(* CODESYS project ATACOMxxxxx_3.0.0.project

Project tree, tasks and I/O mapping:
  Device : HY-TTC 580, TTControl, order no. n/a, version 1.7.1.0
    application Application
      libraries: Standard, * (System); CAA Can Low Level Extern, * (CAA Technical Workgroup); Util, * (System); SysTypes2 Interfaces, * (System); SysTarget, 3.5.5.0 (System); VisuDialogs, * (System); CAA Memory, 3.5.12.0 (CAA Technical Workgroup); Network, 3.5.7.0 (3S - Smart Software Solutions GmbH); lib500, 1.7.1.0 (TTControl); lib500_types, 1.7.1.0 (TTControl); lib500_syscom, 1.7.1.0 (TTControl)
      task _NotificationCallback (externalevent, external event NotificationCallback, priority 0) calls _NotificationCB_PRG
      task _ErrorCallback (externalevent, external event ErrorCallback, priority 1) calls _ErrorCB_PRG
      task CommunicationTask (cyclic, interval t#10ms, priority 31, watchdog t#200ms x 1) calls manageGrCommAndEEPROM, CanCommunication
      task MainTask (cyclic, interval t#10ms, priority 2, watchdog t#200ms x 1) calls MAIN
      Variable lists/
        global variables system
        global variables GVL
        global variables IO
        global variables fieldbus
        global variables par
        global variables CONST
        global variables ERR
        global variables varInput
        global variables display
        global variables ui
        global variables varOutput
      Program logic/
        program _ErrorCB_PRG [ST]
        program _NotificationCB_PRG [ST]
        Tasks/
          program MAIN [ST]: mainLoop, postrun, shutdown, checkParameters, setupCanbus
          program manageGrCommAndEEPROM [ST]: setVariablesToGrComm, initializeGrCommVariables, initializeEepromStructures
          program MachineLogic_PRG [ST]: Cab_C002080
          program CanCommunication [ST]: sendData_to_PC, reciveData_from_PC, initialize
        function initializeCanbus [ST]
        program mngCanbusStatus [ST]: checkCanBusStatus
        program UI_PRG [ST]
        TypeApplication/
          data type Gear9500
      STRUCTURES/
        data type EEPROM_FLAG
        data type CanHandleStatus
        data type MACHINE_MODEL
      Modules/
        IOs/
          Functions/
            program io_module [ST]: instantiateDI, instantiatePWM, instantiatePower, instantiateVOUT, instantiateADC, getInputs, instantiatePWD, initializeIO, instantiateDO, instantiateDIO, instantiatePVG, setOutputs, mngErrors
          program initializeIO [ST]: instantiateAnalogInputs, instantiatePVGOutputs, instantiateDigitalOutputs, instantiateVoltageOutputs, instantiatePWDInputs, instantiatePowerStages, instantiatePWMOutputs, instantiateDigitalInputs
          Types/
            data type pinPWM
            data type type_powerStages
            data type pinADC
            data type type_digitalInputs
            data type pinPVG
            data type type_pwmOutputs
            data type pinPWD
            data type type_voltageOutputs
            data type pinDIO
            data type pwdReadMode
            data type type_digitalOutputs
            data type type_analogInputs
            data type type_pwdInputs
            data type type_pvgOutputs
            data type pin
            data type pinPower
            data type pinVOUT
          global variables sysIO
        COMM/
          Functions/
            program mngCommCan [ST]: mngInit, catchMessages, mngMessage, mngResponse, getsetVarCallback, applyToRamCallback, readAllFromEEPROMCallback, writeToEEPROMCallback, applyToRAM, isVariableValid, initializeVariable
          Types/
            data type grCommVar
            data type grCommAccessRight
            data type grCommVariableStatus
            data type grCommMessageType
            data type grCommEEPROMStatus
          Variable lists/
            global variables grComm
        Canbus/
          Safety interface/
            Tasks/
              program CAN_PRG_SAFE [ST]: exchangeVariables
              program CAN_PRG_UNSAFE [ST]
            Functions/
              program safeSendMessage [ST]
              program safetyCanbusInterface [ST]
              program safeRegisterReceiveMask [ST]
          Variable lists/
            global variables canGVL
            global variables canEVL
          Types/
            data type can
            data type canMessage
            data type canReceiveMask
            data type canBus
          Functions/
            function readMessage [ST]
            program checkReceiveMaskInitialization [ST]
            program registerReceiveMask [ST]
            program sendMessage [ST]
            program initializeCanHandle [ST]
            program checkBusState [ST]
        EEPROM/
          Functions/
            program mngEEPROM [ST]: initEEPROM, mngStep, initializeEepromEntry
          Types/
            Parameters/
              data type HWFW_INFO_TIP
            data type eepromEntry
          Variable lists/
            global variables EEPROM
        Utils/
          program Utils [ST]: decrementUINT, bytesToUInt16, toggle, isNaN, updateValueFiltered, bytesToInt16, decrementUDINT, boolToPWMDutyCycle, linearize, bytesToUReal16, bytesToUDInt32, incrementUINT
        J1939/
          program J1939_PRG [ST]: initReceiveMasks, receiveMessage, parseMessage, sendPGNRequests, mngEngineStatus, redirectToDisplay
          global variables J1939
      visualisation Visualization
    CANs : CANs, TTControl, order no. n/a, version 1.7.1.0
      CAN2 : CAN2, TTControl, order no. n/a, version 1.7.1.0
      CAN3 : CAN3, TTControl, order no. n/a, version 1.7.1.0
      CAN0 : CAN0, TTControl, order no. n/a, version 1.7.1.0
          settings: Baudrate = 250
      CAN1 : CAN1, TTControl, order no. n/a, version 1.7.1.0
      CAN6 : CAN6, TTControl, order no. n/a, version 1.7.1.0
      CAN4 : CAN4, TTControl, order no. n/a, version 1.7.1.0
      CAN5 : CAN5, TTControl, order no. n/a, version 1.7.1.0
    System : System, TTControl, order no. n/a, version 1.7.1.0
        unmapped channels: mode, error, mode, error, mode, error, mode, error, mode, error, mode, error, mode, error, shutdown, error, enable_error_group_0, enable_error_group_1, enable_error_group_2, diag_status, safe_state, error, driver_init_error, UBAT, Terminal_15, WakeUp, Temperature, SSW0, SSW1, SSW2, SSUP0, SSUP1, SSUP2, status, write, boot_error, trigger_error, Powerstage, SSW0, SSW1,
          SSW2, SSUP0, SSUP1, SSUP2, Terminal_15, WakeUp, ExtShutOff0, ExtShutOff1, ExtShutOff2
      Timer_Inputs : TIN, TTControl, order no. n/a, version 1.7.1.0
        Pin 147
          <Empty>
        Pin 122
          <Empty>
        Pin 148
          <Empty>
        Pin 146
          <Empty>
        Pin 124
          <Empty>
        Pin 123
          <Empty>
      Analog_Inputs_2Mode_10V : AIN_2Mode_10V, TTControl, order no. n/a, version 1.7.1.0
        Pin 134
          <Vuoto>
        Pin 109
          <Empty>
        Pin 132
          <Vuoto>
        Pin 131
          <Empty>
        Pin 107
          <Vuoto>
        Pin 110
          <Vuoto>
        Pin 108
          <Empty>
        Pin 133
          <Empty>
      Analog_Inputs_3Mode : AIN_3Mode, TTControl, order no. n/a, version 1.7.1.0
        Pin 129
          <Vuoto>
        Pin 104
          <Vuoto>
        Pin 130
          <Vuoto>
        Pin 105
          <Vuoto>
        Pin 103
          <Vuoto>
        Pin 127
          <Vuoto>
        Pin 106
          <Vuoto>
        Pin 128
          <Empty>
      Digital_Outputs_LS : LSDOUT, TTControl, order no. n/a, version 1.7.1.0
        Pin 239
          <Vuoto>
        Pin 251
          <Vuoto>
        Pin 240
          <Vuoto>
        Pin 252
          <Vuoto>
        Pin 254
          <Vuoto>
        Pin 238
          <Vuoto>
        Pin 253
          <Vuoto>
        Pin 241
          <Vuoto>
      Timer_Inputs_Cur : TIN_Cur, TTControl, order no. n/a, version 1.7.1.0
        Pin 140
          <Empty>
        Pin 117
          <Vuoto>
        Pin 116
          <Empty>
        Pin 139
          <Empty>
        Pin 115
          <Vuoto>
        Pin 141
          <Vuoto>
      Analog_Inputs_2Mode_32V : AIN_2Mode_32V, TTControl, order no. n/a, version 1.7.1.0
        Pin 113
          <Empty>
        Pin 137
          <Empty>
        Pin 136
          <Empty>
        Pin 112
          <Empty>
        Pin 138
          <Empty>
        Pin 114
          <Empty>
        Pin 111
          <Vuoto>
        Pin 135
          <Empty>
      PWM_Outputs : PWM, TTControl, order no. n/a, version 1.7.1.0
        Safety_switch_0 : PWM_SSW0, TTControl, order no. n/a, version 1.7.1.0
          Pin 165
            <Empty>
          Pin 195
            <Vuoto>
          Pin 162
            <Empty>
          Pin 171
            <Vuoto>
          Pin 168
            <Empty>
          Pin 186
            <Empty>
          Pin 183
            <Empty>
          Pin 177
            <Vuoto>
          Pin 180
            <Empty>
          Pin 159
            <Empty>
          Pin 153
            <Vuoto>
          Pin 189
            <Empty>
          Pin 156
            <Empty>
          Pin 192
            <Empty>
        Safety_switch_1 : PWM_SSW1, TTControl, order no. n/a, version 1.7.1.0
          Pin 157
            <Empty>
          Pin 187
            <Empty>
          Pin 154
            <Vuoto>
          Pin 160
            <Empty>
          Pin 178
            <Empty>
          Pin 169
            <Vuoto>
          Pin 166
            <Vuoto>
          Pin 163
            <Empty>
          Pin 184
            <Empty>
          Pin 181
            <Empty>
          Pin 190
            <Vuoto>
          Pin 172
            <Vuoto>
          Pin 193
            <Vuoto>
          Pin 196
            <Vuoto>
        Safety_switch_2 : PWM_SSW2, TTControl, order no. n/a, version 1.7.1.0
          Pin 101
            <Vuoto>
          Pin 125
            <Vuoto>
          Pin 150
            <Vuoto>
          Pin 174
            <Vuoto>
          Pin 102
            <Vuoto>
          Pin 126
            <Vuoto>
          Pin 151
            <Vuoto>
          Pin 175
            <Vuoto>
      Digital_Outputs_HS : HSDOUT, TTControl, order no. n/a, version 1.7.1.0
        Pin 176
          <Vuoto>
        Pin 149
          <Vuoto>
        Pin 158
          <Vuoto>
        Pin 173
          <Vuoto>
        Pin 152
          <Vuoto>
        Pin 155
          <Vuoto>
        Pin 182
          <Vuoto>
        Pin 179
          <Vuoto>
      PVG_Outputs : PVG, TTControl, order no. n/a, version 1.7.1.0
        Pin 161
          <Vuoto>
        Pin 185
          <Vuoto>
        Pin 188
          <Vuoto>
        Pin 164
          <Vuoto>
        Pin 191
          <Vuoto>
        Pin 167
          <Vuoto>
        Pin 194
          <Vuoto>
        Pin 170
          <Vuoto>
  text list GlobalTextList
*)

// Device/Application/STRUCTURES/EEPROM_FLAG
TYPE EEPROM_FLAG : //verificata
STRUCT
	READ: BOOL:= FALSE;
	CHANGED: BOOL:= FALSE;
	WRITE: BOOL:= FALSE;
END_STRUCT
END_TYPE

// Device/Application/Modules/COMM/Types/grCommVar
TYPE grCommVar :
	STRUCT;
		accessRights: grCommAccessRight;
		status: grCommVariableStatus;
		
		pointerToSystemVar: POINTER TO UINT;
		uiLowerValidValue: UINT;
		uiHigherValidValue: UINT;
		uiDefaultValue: UINT;
		
		uiValue: UINT;
	END_STRUCT
END_TYPE

// Device/Application/Modules/COMM/Types/grCommAccessRight
{attribute 'qualified_only'}
{attribute 'strict'}
TYPE grCommAccessRight :
(
	NoAccess := 0,
	ReadOnly := 1,
	ReadWrite := 2
);
END_TYPE

// Device/Application/Modules/COMM/Types/grCommVariableStatus
{attribute 'qualified_only'}
{attribute 'strict'}
TYPE grCommVariableStatus :
(
	Uninitialized:= 0,
	Pristine:= 1,
	ModifiedByRemote:= 2,
	Error:= 3
);
END_TYPE

// Device/Application/Modules/COMM/Types/grCommMessageType
{attribute 'qualified_only'}
{attribute 'strict'}
TYPE grCommMessageType :
(
	ExitCode:= 0,				// Esito di un comando
	
	GetVariable:= 1,			// Get valore di una variabile
	SetVariable:= 2,			// Set valore di una variabile
	HeartRateRequest:= 3,		// Richiesta di heart rate (broadcast)
	LoadFromEEPROM:= 4,			// Leggi parametri da EEPROM
	WriteToEEPROM:= 5,			// Scrivi parametri in RAM sulla EEPROM (rispettando il flag EDIT)
	WriteAllToEEPROM:= 6,		// Scrivi parametri in RAM sulla EEPROM (ignorando il flag EDIT)
	ApplyVariables:= 7,			// Imposta i parametri inviati sulla RAM
	
	ErrorCode:= 255		// Errore
);
END_TYPE

// Device/Application/Modules/IOs/Types/pinPWM
TYPE pinPWM EXTENDS pin :
	STRUCT
		stErrorGetCut: lib500_types.IO_ERRORTYPE;
		wFrequency: WORD:= 100;
		bPolarity: BOOL:= TRUE;
		bDiagMargin: BOOL:= FALSE;
		wFeedbackHighTime: WORD;
		wPeriodFeedback: WORD;
		wCurrent: WORD;
		bCurrentFresh: BOOL;
		wDuty: WORD;
	END_STRUCT
END_TYPE

// Device/Application/Modules/IOs/Types/type_powerStages
TYPE type_powerStages :
STRUCT	
	safetySwitch0: pinPower;	
	safetySwitch1: pinPower;	
	safetySwitch2: pinPower;
	powerStage: pinPower;
	sensorSupply0: pinPower;
	sensorSupply1: pinPower;
	sensorSupply2: pinPower;
END_STRUCT
END_TYPE

// Device/Application/Modules/IOs/Types/pinADC
TYPE pinADC EXTENDS pin :
	STRUCT		
		stADCType: lib500_types.IO_ADC_TYPE;
		stADCRange: lib500_types.IO_ADC_RANGE;
		stADCSensorSupply: lib500_types.IO_SENSOR_SUPPLY;
		dwValue: DWORD;
		bValueFresh: BOOL;
	END_STRUCT
END_TYPE

// Device/Application/Modules/COMM/Types/grCommEEPROMStatus
{attribute 'qualified_only'}
{attribute 'strict'}
TYPE grCommEEPROMStatus :
(
	Idle:= 0,
	BeginRead:= 1,
	Reading:= 2,
	BeginWrite:= 3,
	Writing
);
END_TYPE

// Device/Application/Modules/IOs/Types/type_digitalInputs
TYPE type_digitalInputs :
STRUCT	
	fuelReserve_p127: pinDIO;
	alternatorD_p111: pinDIO;
	gearSelectorFwInching_p135: pinDIO;
	gearSelectorFirstSlow_p112: pinDIO;
	gearSelectorBwInching_p136: pinDIO;
	gearSelectorSecondFast_p113: pinDIO;
	inchingSwitch_p137: pinDIO;
	compressedAirSwitch_p114: pinDIO;
	safetySwitch_p138: pinDIO;
	
	parkingBrakeLamp_p140: pinDIO;
	airPressureLowLamp_p177: pinDIO;
	transOilOvertempLamp_p156: pinDIO;
	brakeFluidLowLamp_p180: pinDIO;
	coolantLevelLow_p159: pinDIO;
	
	engineStartK50_p117: pinDIO;
	seatSwitch_p146: pinDIO;
	forwardSwitch_p123: pinDIO;
	backwardSwitch_p147: pinDIO;
	neutralSwitch_p124: pinDIO;
	
	turtleSwitch_p161: pinDIO;
	positionLightsSwitch_p185: pinDIO;
	lowBeamLightsSwitch_p188: pinDIO;
	highBeamFlashLightsSwitch_p164: pinDIO;
	highBeamLightsSwitch_p116: pinDIO;
	leftBlinkerSwitch_p191: pinDIO;
	rightBlinkerSwitch_p167: pinDIO;
	hazardSwitch_p194: pinDIO;
	parkingBrakeSwitchOptional_p170: pinDIO;
	
	speedLimiterSwitch_p129: pinDIO;
	
	gearShiftUp_p122: pinDIO;
	gearShiftDown_p148: pinDIO;
	autoDetect9500_p238: pinDIO;
	
	

	
	input_115: pinDIO;
	input_116: pinDIO;
	input_117: pinDIO;
	input_122: pinDIO;
	input_123: pinDIO;
	input_124: pinDIO;
	input_139: pinDIO;
	input_140: pinDIO;
	input_141: pinDIO;
	input_146: pinDIO;
	input_147: pinDIO;
	input_148: pinDIO;
	input_161: pinDIO;
	input_164: pinDIO;
	input_167: pinDIO;
	input_170: pinDIO;
	input_185: pinDIO;
	input_188: pinDIO;
	input_191: pinDIO;
	input_194: pinDIO;
	
	
	
	
END_STRUCT
END_TYPE

// Device/Application/Modules/IOs/Types/pinPVG
TYPE pinPVG EXTENDS pin :
	STRUCT
		stGetVoltageError: lib500_types.IO_ERRORTYPE;
		wValue: WORD := 5000;
		uiReadVoltage: UINT := 0;
		bVoltageFresh: BOOL := FALSE;
	END_STRUCT
END_TYPE

// Device/Application/Modules/Canbus/Types/can
TYPE can :
	STRUCT
			
		bInitialized: BOOL:= FALSE;	
		usiChannel: USINT:= 0;
		uiBaudrateKbps: UINT:= 0;
	
		driver: CL2.CAA.HANDLE;
		initializeError: CL2.ERROR;
		transmitError: CL2.ERROR;
		busStatus: CL2.BUSSTATE;
		
		receiveMessageHandle: CL2.CAA.HANDLE := CL2.CAA.gc_hINVALID;
		pointerToData: POINTER TO CL2.CL2I.DATA;
		messageLeft : CL2.CAA.COUNT;
		
		uiMessageCount: INT:=0;
		byaReceiveBuffer: ARRAY [0..7] OF BYTE;				
		byaTransmitBuffer: ARRAY [0..7] OF BYTE;						
		
	END_STRUCT
END_TYPE

// Device/Application/Modules/IOs/Types/type_pwmOutputs
TYPE type_pwmOutputs :
STRUCT
	turtleBtnBacklight_p168: pinPWM;
	hazardBtnBacklight_p190: pinPWM;
END_STRUCT
END_TYPE

// Device/Application/Modules/Canbus/Types/canMessage
TYPE canMessage :
	STRUCT
		udiId: UDINT:= 0;
		bExtended: BOOL:= FALSE;
		byLength: BYTE:= 8;
		byaData: ARRAY [0..7] OF BYTE;
	END_STRUCT
END_TYPE

// Device/Application/Modules/Canbus/Types/canReceiveMask
TYPE canReceiveMask :
	STRUCT
		bActive: BOOL:= FALSE;
		bInitialized: BOOL:= FALSE;
		udiId: UDINT:= 0;
		stCAAMask: CL2.CAA.HANDLE:= CL2.CAA.gc_hINVALID;	
		stMessagesLeft: CL2.CAA.COUNT;	
		udiCobIdMask: UDINT:= 16#1FFFFFFF;
	END_STRUCT
END_TYPE

// Device/Application/Modules/Canbus/Types/canBus
TYPE canBus :
	STRUCT
		bActive: BOOL:= FALSE;
		stChannel: can;
		staReceiveMasks: ARRAY[0..canGVL.iReceiveMaskCount-1] OF canReceiveMask;
		stTransmitBuffer: ARRAY[0..canGVL.iTransmitBufferSize-1] OF canMessage;
	END_STRUCT
END_TYPE

// Device/Application/Modules/IOs/Types/pinPWD
TYPE pinPWD EXTENDS pin :
	STRUCT
		stGetVoltageError: lib500_types.IO_ERRORTYPE;
		stIncSetError: lib500_types.IO_ERRORTYPE;
		pwdMode: lib500_types.IO_PWD_INC_MODE;
		wCountInit: WORD:= 32767;
		wCount: WORD;
		wCountZero: WORD;
		uiVoltage: UINT;
		bChannelA: BOOL;
		bChannelB: BOOL;
		readMode: pwdReadMode;
		pulseSamples: lib500_types.IO_PWD_PULSE_SAMPLES;
		dwFrequencyHz: DWORD;
		dwPulseWidth: DWORD;
		pulseMode: lib500_types.IO_PWD_PULSE_MODE;
		freqMode: lib500_types.IO_PWD_FREQ_MODE;
		byCaptureCount: BYTE;
		bVoltageFresh: BOOL;
		bSetIncrementCount: BOOL:= FALSE;
	END_STRUCT
END_TYPE

// Device/Application/Modules/IOs/Types/type_voltageOutputs
TYPE type_voltageOutputs :
STRUCT
	// dummy: pinVOUT;
END_STRUCT
END_TYPE

// Device/Application/STRUCTURES/CanHandleStatus
TYPE CanHandleStatus :
	STRUCT
		uidFreeMessagesInPoll: UDINT:= 0;
		uidMessagesInElabQueue: UDINT:= 0;
	END_STRUCT
END_TYPE

// Device/Application/Modules/IOs/Types/pinDIO
TYPE pinDIO EXTENDS pin :
	STRUCT
		bValue: BOOL:= FALSE;
		wCurrent: WORD;
		bCurrentFresh: BOOL;
		stErrorGetCut: lib500_types.IO_ERRORTYPE;
	END_STRUCT
END_TYPE

// Device/Application/Modules/IOs/Types/pwdReadMode
{attribute 'qualified_only'}
{attribute 'strict'}
TYPE pwdReadMode :
(
	incremental := 0,
	complex
);
END_TYPE

// Device/Application/Modules/IOs/Types/type_digitalOutputs
TYPE type_digitalOutputs :
STRUCT				 
	lampeggiante_p183: pinDIO;
	workLights_p186: pinDIO;
	airCompressorRelay_p162: pinDIO;
	dashboardBacklight_p189: pinDIO;
	workModeActiveDpfLamp_p165: pinDIO;
	forwardGearEV_p192: pinDIO;

	backwardGearEV_p193: pinDIO;
		
	highBeamLights_p149: pinDIO;
	highBeamLights_p173: pinDIO;
	
	lowBeamLights_p152: pinDIO;
	lowBeamLights_p176: pinDIO;
	
	positionLights_p155: pinDIO;
	positionLights_p179: pinDIO;
	
	inchingBrakeEV_p171: pinDIO;
	parkingBrakeEV_p154: pinDIO;
	pneumaticParkBrakeEV_p178: pinDIO;
	rightBlinker_p157: pinDIO;
	leftBlinker_p181: pinDIO;
	reverseLight_p160: pinDIO;
	neutralGear_p254: pinDIO;
	reverseBuzzer_p184: pinDIO;
	
	inchingLamp_p163: pinDIO;
	daytimeLights_p187: pinDIO;
	displayK15_p166: pinDIO;
	
	slowGearEV_p195: pinDIO;//gearEvC_p195: pinDIO;
	gearEvD_p169: pinDIO;
	gearEvE_p196: pinDIO;
	
	output_149: pinDIO;
	output_150: pinDIO;
	output_152: pinDIO;
	output_153: pinDIO;
	output_154: pinDIO;
	output_155: pinDIO;
	output_156: pinDIO;
	output_157: pinDIO;
	output_158: pinDIO;
	output_159: pinDIO;
	output_173: pinDIO;
	output_174: pinDIO;
	output_176: pinDIO;
	output_177: pinDIO;
	output_178: pinDIO;
	output_179: pinDIO;
	output_180: pinDIO;
	output_181: pinDIO;
	output_182: pinDIO;
	output_183: pinDIO;
END_STRUCT
END_TYPE

// Device/Application/Modules/IOs/Types/type_analogInputs
TYPE type_analogInputs :
STRUCT
	ecuK15_p207: pinADC;
	fuelTankGauge_p103: pinADC;	
	pneumaticTankGauge_p104: pinADC;
	shiftOilGauge_p128: pinADC;	
	
	speedLimiterReduction_p251: pinADC;	
END_STRUCT
END_TYPE

// Device/Application/Modules/IOs/Types/type_pwdInputs
TYPE type_pwdInputs :
STRUCT
	//speedSensor_p115: pinPWD;
	transmissionShaftSensor5000_p175: pinPWD;
	transmissionShaftSensor7500_p151: pinPWD;
END_STRUCT
END_TYPE

// Device/Application/Modules/IOs/Types/type_pvgOutputs
TYPE type_pvgOutputs :
STRUCT
	//_p161: pinPWD;
END_STRUCT
END_TYPE

// Device/Application/Modules/IOs/Types/pin
TYPE pin :
	STRUCT
		bInitialized: BOOL:= FALSE;
		stInitError: lib500_types.IO_ERRORTYPE;
		stError: lib500_types.IO_ERRORTYPE;
		byChannel: BYTE;
		byPullType: BYTE;
		byMinTTCModel: BYTE:= 0;
		byResetCount: BYTE:= 0;
	END_STRUCT
END_TYPE

// Device/Application/Modules/IOs/Types/pinPower
TYPE pinPower EXTENDS pin :
	STRUCT
		mode: lib500_types.IO_POWER_STATE;
	END_STRUCT
END_TYPE

// Device/Application/Modules/EEPROM/Types/eepromEntry
TYPE eepromEntry :
	STRUCT
		wAddress: WORD;
		pData: POINTER TO BYTE;
		wSize: WORD;
	END_STRUCT
END_TYPE

// Device/Application/Modules/EEPROM/Types/Parameters/HWFW_INFO_TIP
TYPE HWFW_INFO_TIP :
	STRUCT		
		PASSWORD_LEVEL_0: UINT:= 0;
		PASSWORD_LEVEL_1: UINT:= 1234;		
	END_STRUCT
END_TYPE

// Device/Application/Modules/IOs/Types/pinVOUT
TYPE pinVOUT EXTENDS pin :
	STRUCT
		wOutputVoltageMv: WORD:= 0;
	END_STRUCT
END_TYPE

// Device/Application/STRUCTURES/MACHINE_MODEL
{attribute 'qualified_only'}
{attribute 'strict'}
TYPE MACHINE_MODEL :
(
	ATA_5000 := 0,
	ATA_7500,
	ATA_9500
);
END_TYPE

// Device/Application/Program logic/TypeApplication/Gear9500
{attribute 'qualified_only'}
{attribute 'strict'}
TYPE Gear9500 :
(
	GEAR_1ST := 1,
	GEAR_2ND,
	GEAR_3RD,
	GEAR_4TH
);
END_TYPE

// Device/Application/Modules/COMM/Variable lists/grComm
{attribute 'qualified_only'}

(* User code configurable settings *)
VAR_GLOBAL CONSTANT
	uiProtocolMessageID : UINT:=16#7F7;
	uiProtocolVirtualNode : UINT:=16#3;	
	uiVariablesMaxIndex: UINT:= 100;    // Reduce this value if you have low memory issues
END_VAR



(* User code accessible status variables *)
VAR_GLOBAL  			
	bCommunicationActive: BOOL:=FALSE;			// Indicates that a communication is running
	bTriggerReadFromEEPROM: BOOL:= TRUE;		// If active user code should read variables from EEPROM and store their value in grComm.staVariables
	bTriggerApplyToRAM: BOOL:= FALSE;			// If active user code should set its system values from grComm.staVariables
	bTriggerWriteToEEPROM: BOOL:= FALSE;		// If active user code should write to EEPROM only the modified variable's values from grComm.staVariables
	bTriggerWriteAllToEEPROM: BOOL:= FALSE;		// If active user code should write to EEPROM all the variable's values from grComm.staVariables
END_VAR


(* Internal logic variables *)
VAR_GLOBAL
	staVariables: ARRAY[1..uiVariablesMaxIndex] OF grCommVar;	
END_VAR

(* Internal logic defines *)
VAR_GLOBAL CONSTANT	
	COMM_TIMER_RLD: UINT:= 1000;
	LIB_VERSION_CODE: BYTE:= 0;		
	
	// Exit code viene messo nel campo ADDRESS se TYPE == EXIT_CODE
	EXIT_CODE_ERROR: UINT:= 0;
	EXIT_CODE_OK: UINT:= 1;

END_VAR

// Device/Application/Variable lists/system
{attribute 'qualified_only'}
VAR_GLOBAL CONSTANT	
	FWV_PRIMARIA: BYTE:=0;
	FWV_SECONDARIA: BYTE:=0;
	FWV_BUGFIX: BYTE:=0;	
END_VAR

VAR_GLOBAL	
	xFirstCycle: BOOL:= TRUE;
	
	machineModel: MACHINE_MODEL;
	
	fwVMergedPrimarySecondary: UINT:= (FWV_PRIMARIA * 256) OR FWV_SECONDARIA;
	fwVMergedRevisionBugfix: UINT:= FWV_BUGFIX;
	bHasAlarms: BOOL:= FALSE;	
	
	matricolaL: UINT:= 0;
	matricolaH: UINT:= 0;
	
	bParametersReady: BOOL:= FALSE;	
	systemAlarms: UINT:= 0;
	
	xHazardStatus: BOOL:= FALSE;
	xParkingBrakeActive: BOOL:= FALSE;
	xParkingBrakeLampInputActive: BOOL:= FALSE;
	xInchingModeActive: BOOL:= FALSE;
	
	byActiveGear: BYTE:= 0;  (* 1-EvMarciaLentaAttiva, 2-EvMarciaLentaDisattiva NoInching, 3-Inching  *)
	byDirection: BYTE:= 0;  (* 0- ferma, 1-avanti, 2 indietro *)
	byFuelPercent: BYTE;
	
	xSeatStatus: BOOL;
	rFuelLevelFiltered: REAL;
	udiInchingAlertTimerMs: UDINT;
	
	rSpeedKmph: REAL;
	xIncorrectStart: BOOL;
END_VAR

// Device/Application/Variable lists/GVL
{attribute 'qualified_only'}
VAR_GLOBAL
	MODELLO_CENTRALINA: BYTE;
	fwVersion: ARRAY[0..2] OF BYTE:= [3, 0, 0];  // versione di cenrtralina 3.0.0
	
	xAllowSystemShutdown: BOOL;
	xDPFRegenerationRequestInput: BOOL;	
	xSpeedLimitStatus: BOOL:= FALSE;
END_VAR

// Device/Application/Variable lists/IO
{attribute 'qualified_only'}
VAR_GLOBAL
	xECUK15: BOOL;
	
	xSpeedLimFromAdc: BOOL;
END_VAR

// Device/Application/Modules/Canbus/Variable lists/canGVL
{attribute 'qualified_only'}

VAR_GLOBAL CONSTANT	
	iBusCount: INT:= 10;
	iTransmitBufferSize: INT:= 50;
	iReceiveMaskCount: INT:= 50;
END_VAR

VAR_GLOBAL
	busses: ARRAY[0..iBusCount-1] OF canBus;
END_VAR

// Device/Application/Variable lists/fieldbus
{attribute 'qualified_only'}
VAR_GLOBAL CONSTANT
	iCanbusCount: INT:= 4;
	uiaCanBaudrates: ARRAY[0..9] OF UINT:= [500, 250, 250, 0, 0, 0, 0, 0, 0, 0];
END_VAR

VAR_GLOBAL
	can: ARRAY [0..9] OF canBus;
	
	bCanbusInitialized: BOOL:= FALSE;
END_VAR

// Device/Application/Variable lists/par
{attribute 'qualified_only'}
VAR_GLOBAL
	stHwFwInfo: HWFW_INFO_TIP;
END_VAR

// Device/Application/Variable lists/CONST
{attribute 'qualified_only'}
VAR_GLOBAL	
	CANBUS_MAX_READS_PER_CYCLE: BYTE:= 10;
	CANBUS_MIN_FREE_POLL: BYTE:= 30;
	CANBUS_MAX_RX_QUEUE: BYTE:= 15;
END_VAR

// Device/Application/Modules/IOs/sysIO
{attribute 'qualified_only'}
VAR_GLOBAL
	bIOInstantiated: BOOL:= FALSE;
	bIOInitialized: BOOL:= FALSE;

	digitalInput: type_digitalInputs;
	analogInput: type_analogInputs;
	pwdInput: type_pwdInputs;
	pvgOutput: type_pvgOutputs;
	
	digitalOutput: type_digitalOutputs;
	powerStage: type_powerStages;
	pwmOutput: type_pwmOutputs;
	voltageOutput: type_voltageOutputs;
END_VAR

// Device/Application/Modules/Canbus/Variable lists/canEVL
(* THIS EVL IS AUTOGENERATED. DO NOT MODIFY THESE ATTRIBUTES. *)
{attribute 'location' := '16#800' }
{attribute 'linkalways'}
{attribute 'qualified_only'}
VAR_GLOBAL	
	bHasChanges: BOOL:= FALSE;
	bChannelsHasChanges: BOOL:= FALSE;
	bTransmitBuffersHasChanges: BOOL:= FALSE;
	bMasksHasChanges: BOOL:= FALSE;
	busses: ARRAY[0..canGVL.iBusCount-1] OF canBus;
END_VAR

// Device/Application/Modules/EEPROM/Variable lists/EEPROM
{attribute 'qualified_only'}

(* User code accessible status indicators *)
VAR_GLOBAL
	bTriggerReadAll: BOOL:= FALSE;
	
	bEEPROMInitialized: BOOL := FALSE;
	bReadFromEEPROM: BOOL := TRUE;
	bWriteAllToEEPROM: BOOL:= FALSE;
END_VAR


(* Internal logic *)
VAR_GLOBAL CONSTANT	
	iEepromEntriesCount: INT:= 160;
END_VAR
VAR_GLOBAL	
	staAllEntries: ARRAY[0..iEepromEntriesCount-1] OF eepromEntry; // On TTC-500 series EEPROM is 64KB. Each structure has 400 byte of space reserved
END_VAR

// Device/Application/Variable lists/ERR
{attribute 'qualified_only'}
VAR_GLOBAL
	xInputPins: BOOL;
	xOutputPins: BOOL;
	xInitializePins: BOOL;
	xCanbusHeavy: BOOL;
END_VAR

// Device/Application/Variable lists/varInput
{attribute 'qualified_only'}
VAR_GLOBAL
	xInput_1: BOOL;
	xInput_2: BOOL;
	xInput_3: BOOL;
	xInput_4: BOOL;
	xInput_5: BOOL;
	xInput_6: BOOL;
	xInput_7: BOOL;
	xInput_8: BOOL;
	xInput_9: BOOL;
	xInput_10: BOOL;
	xInput_11: BOOL;
	xInput_12: BOOL;
	xInput_13: BOOL;
	xInput_14: BOOL;
	xInput_15: BOOL;
	xInput_16: BOOL;
	xInput_17: BOOL;
	xInput_18: BOOL;
	xInput_19: BOOL;
	xInput_20: BOOL;
END_VAR

// Device/Application/Variable lists/display
{attribute 'qualified_only'}
VAR_GLOBAL
	xLampeggianteOffStatus: BOOL:= FALSE;
	xWorkLightStatus: BOOL:= FALSE;
	xDRLOffStatus: BOOL:= FALSE;
	xSpeedLimitRequest: BOOL:= FALSE;
	
	xInput1, xInput2, xInput3, xInput4, xInput5, xInput6, xInput7, xInput8: BOOL;
END_VAR

// Device/Application/Variable lists/ui
{attribute 'qualified_only'}
VAR_GLOBAL
	xBlinker_100ms: BOOL;
	xBlinker_500ms: BOOL;
END_VAR

// Device/Application/Modules/J1939/J1939
{attribute 'qualified_only'}
VAR_GLOBAL
	byECUNodeId: BYTE:= 16#10;
	xEngineOnline: BOOL:= FALSE;
	xSendPGNRequest: BOOL:= FALSE;
	xRedirectMessages: BOOL:= FALSE;
	
	// valori in arrivo dal bus
	iTorquePercent: INT;
	uiEngineSpeedRpm: UINT;
	uiMinutesRunWhileMILAct: UINT;
	lrEngineTotalFuelUsedLiters: LREAL;
	rEngineFuelRateLph: REAL;
	byBarometricPressureKPa: BYTE;
	iAmbientAirTemperatureDegC: INT;
	iEngineIntakeAirTemperatureDegC: INT;
	uiOilPressureKPa: UINT;
	byCoolantLevelPerc: BYTE;
	iEngineCoolantTempDegC: INT;
	iEngineFuelTempDegC: INT;
	iAftertreatmentDPFIntakeGasTempDegC: INT;
	rBatteryPotentialV: REAL;
	byEngineStartEnable: BYTE;
	rEngineTotalIdleHours: REAL;
	byAftertreatmentEngineSpeedIncreaseRequest: BYTE;
	byEngineWaitToStartLamp: BYTE;
	byEngineIdleShutdownStatus: BYTE;
	byEngineIdleShutdownAlert: BYTE;
	byServiceComponentId1: BYTE;
	byServiceComponentId2: BYTE;
	byServiceComponentId3: BYTE;
	iServiceDelayHours: INT;
	rEngineTotalOperationHours: REAL;
	byDPFFilterLamp: BYTE;
	byAftertreatmentDPFActiveRegeneration: BYTE;
	byAftertreatmentDPFFilterStatus: BYTE;
	byDPFActiveRegenerationInhibitedDueSwitch: BYTE;
	byDPFActiveRegenerationInhibitedDueTmpSysLock: BYTE;
	byDPFActiveRegenerationInhibitedDuePermSysLock: BYTE;
	
	
	byWarningIndicator: BYTE;	
	byWarningIndicatorFlash: BYTE;
	byShutdownIndicator: BYTE;
	byEngineProtectIndicator: BYTE;
	byEngineProtectIndicatorFlash: BYTE;
	byEmissionSystemMalfunctionIndicator: BYTE;
	byEmissionSystemMalfunctionIndicatorFlash: BYTE;	
	
	
	// trouble codes
	DM1_SPN: ULINT;
	DM1_FMI: UINT;
	DM1_OC: UINT;
	
	
	// valori calcolati
	xEngineRunning: BOOL;
	xEngineDPFRegenRequest: BOOL;
	xEngineDPFRegenActive: BOOL;
	xLowOilPressure: BOOL;
	xEngineLamp: BOOL;
	xEngineLampRed: BOOL;
	byRegenerationStatus: BYTE;
	
	
END_VAR

// Device/Application/Variable lists/varOutput
{attribute 'qualified_only'}
VAR_GLOBAL
	xOutput_1: BOOL;
	xOutput_2: BOOL;
	xOutput_3: BOOL;
	xOutput_4: BOOL;
	xOutput_5: BOOL;
	xOutput_6: BOOL;
	xOutput_7: BOOL;
	xOutput_8: BOOL;
	xOutput_9: BOOL;
	xOutput_10: BOOL;
	xOutput_11: BOOL;
	xOutput_12: BOOL;
	xOutput_13: BOOL;
	xOutput_14: BOOL;
	xOutput_15: BOOL;
	xOutput_16: BOOL;
	xOutput_17: BOOL;
	xOutput_18: BOOL;
	xOutput_19: BOOL;
	xOutput_20: BOOL;
END_VAR

// Device/Application/Program logic/_NotificationCB_PRG
PROGRAM _NotificationCB_PRG
VAR
	diag_state : lib500_types.DIAG_STATETYPE := lib500_types.DIAG_STATETYPE.DIAG_STATE_DISABLED;
	watchdog_state : lib500_types.DIAG_WD_STATETYPE := lib500_types.DIAG_WD_STATETYPE.DIAG_WD_STATE_UNKNOWN;
	error : lib500_types.DIAG_ERRORCODE := (error_code := lib500_types.DIAG_ERRORTYPE.DIAG_E_NOERROR, 
                                            device_num := lib500_types.DIAG_DEVICETYPE.DIAG_DEV_NONE,
                                            faulty_value := 0);
	return_code : lib500_types.IO_ERRORTYPE := lib500_types.IO_ERRORTYPE.IO_E_UNKNOWN;
	
	call_count : UDINT := 0;
END_VAR

(* get the reason for the notification callback *)
return_code := lib500.DIAG_CDS_GetNotificationReason(ADR(diag_state), 
                                                     ADR(watchdog_state),
                                                     ADR(error));

(* custom handler code can be placed here *)

(* increment call count *)
call_count := call_count + 1;

END_PROGRAM

// Device/Application/Program logic/_ErrorCB_PRG
PROGRAM _ErrorCB_PRG
VAR
	diag_state : lib500_types.DIAG_STATETYPE := lib500_types.DIAG_STATETYPE.DIAG_STATE_DISABLED;
	watchdog_state : lib500_types.DIAG_WD_STATETYPE := lib500_types.DIAG_WD_STATETYPE.DIAG_WD_STATE_UNKNOWN;
	error : lib500_types.DIAG_ERRORCODE := (error_code := lib500_types.DIAG_ERRORTYPE.DIAG_E_NOERROR, 
                                            device_num := lib500_types.DIAG_DEVICETYPE.DIAG_DEV_NONE,
                                            faulty_value := 0);
	return_code : lib500_types.IO_ERRORTYPE := lib500_types.IO_ERRORTYPE.IO_E_UNKNOWN;
	
	reaction : lib500_types.DIAG_REACTION := lib500_types.DIAG_REACTION.DIAG_ERR_SAFESTATE;
	
	call_count : UDINT := 0;
END_VAR

(* get the reason for the error callback *)
return_code := lib500.DIAG_CDS_GetErrorReason(ADR(diag_state), 
                                              ADR(watchdog_state),
                                              ADR(error));

(* custom handler code can be placed here *)

(* the choices for the reactions are:
   -> lib500_types.DIAG_REACTION.DIAG_ERR_NOACTION
   -> lib500_types.DIAG_REACTION.DIAG_ERR_SAFESTATE
   -> lib500_types.DIAG_REACTION.DIAG_ERR_DISABLE_SSW0
   -> lib500_types.DIAG_REACTION.DIAG_ERR_DISABLE_SSW1
   -> lib500_types.DIAG_REACTION.DIAG_ERR_DISABLE_SSW2
   -> lib500_types.DIAG_REACTION.DIAG_ERR_DISABLE_HS00
   -> lib500_types.DIAG_REACTION.DIAG_ERR_DISABLE_HS01
   -> lib500_types.DIAG_REACTION.DIAG_ERR_DISABLE_HS02
   -> lib500_types.DIAG_REACTION.DIAG_ERR_DISABLE_HS03
   -> lib500_types.DIAG_REACTION.DIAG_ERR_DISABLE_HS04
   -> lib500_types.DIAG_REACTION.DIAG_ERR_DISABLE_HS05
   -> lib500_types.DIAG_REACTION.DIAG_ERR_DISABLE_HS06
   -> lib500_types.DIAG_REACTION.DIAG_ERR_DISABLE_HS07
   
   it's also possible to combine (binary-or) reactions, like:
   -> lib500_types.DIAG_REACTION.DIAG_ERR_DISABLE_SSW0 OR 
      lib500_types.DIAG_REACTION.DIAG_ERR_DISABLE_SSW1
*)

(* pass the error reaction to the DIAG system *)
lib500.DIAG_CDS_SetErrorReaction(reaction);

(* increment call count *)
call_count := call_count + 1;

END_PROGRAM

// Device/Application/Program logic/Tasks/manageGrCommAndEEPROM
PROGRAM manageGrCommAndEEPROM
VAR
	bGrCommInitialized: BOOL:= FALSE;
	bEepromStructuresInitialized: BOOL:= FALSE;
	uiDummy: UINT:= 0;
END_VAR

(* 
*  You must respect this priorities to allow grComm to 
*  always give a consistent value to the variables 
*)
IF NOT bEepromStructuresInitialized THEN
	bEepromStructuresInitialized:= initializeEepromStructures();
	
ELSIF NOT bGrCommInitialized THEN
	bGrCommInitialized:= initializeGrCommVariables();
	
ELSIF grcomm.bTriggerReadFromEEPROM THEN
	EEPROM.bReadFromEEPROM:= TRUE;
	grcomm.bTriggerReadFromEEPROM:= FALSE;

ELSIF EEPROM.bReadFromEEPROM THEN
	mngEEPROM();
	bGrCommInitialized:= EEPROM.bReadFromEEPROM; 							// when reading has ended, triggers initialization 
	IF NOT EEPROM.bReadFromEEPROM THEN system.bParametersReady:= TRUE; END_IF	// when reading has ended, activate parameters ready flag

ELSIF grcomm.bTriggerApplyToRAM THEN
	mngCommCan.applyToRAM();
	grcomm.bTriggerApplyToRAM:= FALSE;

ELSIF (grcomm.bTriggerWriteToEEPROM OR grcomm.bTriggerWriteAllToEEPROM) THEN
	EEPROM.bWriteAllToEEPROM:= TRUE;
	grcomm.bTriggerWriteToEEPROM:= FALSE;
	grcomm.bTriggerWriteAllToEEPROM:= FALSE;

ELSIF EEPROM.bWriteAllToEEPROM THEN
	mngEEPROM();
	EEPROM.bReadFromEEPROM:= EEPROM.bReadFromEEPROM; // when reading has ended, triggers read from eeprom
	
ELSE
	setVariablesToGrComm();
	mngCommCan(stCanbus:= fieldbus.can[1]);
END_IF

METHOD PRIVATE setVariablesToGrComm
VAR
	uiVarIterator: UINT;
END_VAR
FOR uiVarIterator:= 1 TO grComm.uiVariablesMaxIndex BY 1 DO
	IF mngCommCan.isVariableValid(grComm.staVariables[uiVarIterator]) AND (grComm.staVariables[uiVarIterator].status <> grCommVariableStatus.ModifiedByRemote) THEN
		grComm.staVariables[uiVarIterator].uiValue:= grComm.staVariables[uiVarIterator].pointerToSystemVar^;
	END_IF
END_FOR
END_METHOD

METHOD PRIVATE initializeGrCommVariables : BOOL
VAR_INPUT
END_VAR
(* user code should setup the desired addresses like this 
*      grComm.staVariables[ <NETWORK_ADDR> ]:= mngCommCan.initializeVariable(
*										pointerToSystemVar:= ADR( <SYS_VARIABLE> ),
*										accessRights:= grCommAccessRight.ReadOnly,
*										uiDefaultValue:= x,
*										uiLowerValidValue:= y,
*										uiHigherValidValue:= z
*									);
*  use the variable address as the array index.
*  You can make the code more readable passing the arguments without naming it
*)		
		
grComm.staVariables[2]:= 		mngCommCan.initializeVariable(ADR(uiDummy),		grCommAccessRight.ReadOnly, 1, 0, 16#FFFF);
grComm.staVariables[3]:= 		mngCommCan.initializeVariable(ADR(uiDummy),		grCommAccessRight.ReadOnly, 1, 0, 16#FFFF);
grComm.staVariables[4]:= 		mngCommCan.initializeVariable(ADR(uiDummy),		grCommAccessRight.ReadOnly, 1, 0, 16#FFFF);

grComm.staVariables[5]:= 		mngCommCan.initializeVariable(ADR(system.fwVMergedPrimarySecondary),		grCommAccessRight.ReadOnly, 1, 0, 16#FFFF);
grComm.staVariables[6]:= 		mngCommCan.initializeVariable(ADR(system.fwVMergedRevisionBugfix),			grCommAccessRight.ReadOnly, 1, 0, 16#FFFF);
grComm.staVariables[7]:= 		mngCommCan.initializeVariable(ADR(system.matricolaH),						grCommAccessRight.ReadOnly, 1, 0, 16#FFFF);
grComm.staVariables[8]:= 		mngCommCan.initializeVariable(ADR(system.matricolaL),						grCommAccessRight.ReadOnly, 1, 0, 16#FFFF);
grComm.staVariables[9]:= 		mngCommCan.initializeVariable(ADR(system.systemAlarms),						grCommAccessRight.ReadWrite, 0, 0, 16#FFFF);

grComm.staVariables[16#0A]:=	mngCommCan.initializeVariable(ADR(par.stHwFwInfo.PASSWORD_LEVEL_0),		grCommAccessRight.ReadWrite, 0, 	0, 16#FFFF);
grComm.staVariables[16#0B]:=	mngCommCan.initializeVariable(ADR(par.stHwFwInfo.PASSWORD_LEVEL_1),		grCommAccessRight.ReadWrite, 1234, 	0, 16#FFFF);


initializeGrCommVariables:= TRUE;
END_METHOD

METHOD PRIVATE initializeEepromStructures : BOOL
VAR_INPUT
END_VAR
mngEEPROM.initializeEepromEntry(wAddress:= 16#0000, pData:= ADR(par.stHwFwInfo), wSize:= SIZEOF(par.stHwFwInfo));

initializeEepromStructures:= TRUE;
END_METHOD

END_PROGRAM

// Device/Application/Modules/EEPROM/Functions/mngEEPROM
PROGRAM mngEEPROM
VAR	
	eepromErrorCode : lib500_types.IO_ERRORTYPE := lib500_types.IO_ERRORTYPE.IO_E_OK;
	eepromStatus : lib500_types.IO_ERRORTYPE := lib500_types.IO_ERRORTYPE.IO_E_OK;
	eepromLoopStep : INT:=0;
	
	eepromBusy: BOOL:= FALSE;
	iEntryCursor: INT:= 0;
END_VAR

IF NOT EEPROM.bEEPROMInitialized THEN
	initEEPROM();

ELSIF (NOT EEPROM.bReadFromEEPROM) AND (NOT EEPROM.bWriteAllToEEPROM) THEN
	RETURN;
	
ELSE		
	
	mngStep(uiAddress:= EEPROM.staAllEntries[eepromLoopStep].wAddress, 
			bRead:= EEPROM.bReadFromEEPROM, 
			pData:= EEPROM.staAllEntries[eepromLoopStep].pData, 
			wLength:= EEPROM.staAllEntries[eepromLoopStep].wSize);

	(* eepromLoopStep is incremented by mngStep function *)			
	IF (EEPROM.staAllEntries[eepromLoopStep].pData = 0) THEN				
		EEPROM.bReadFromEEPROM:= FALSE;
		EEPROM.bWriteAllToEEPROM:= FALSE;
		eepromLoopStep:= 0;	
	END_IF
	
END_IF

ACTION initEEPROM:
eepromErrorCode := lib500.IO_EEPROM_Init();		
eepromStatus := lib500.IO_EEPROM_GetStatus();
EEPROM.bEEPROMInitialized:= (eepromStatus = lib500_types.IO_ERRORTYPE.IO_E_OK);
END_ACTION

METHOD mngStep
VAR_INPUT
	bRead: BOOL;
	uiAddress: UINT;
	pData: POINTER TO BYTE;
	wLength: WORD;
END_VAR
IF NOT eepromBusy THEN	
	eepromErrorCode := lib500.IO_EEPROM_GetStatus();
	IF (eepromErrorCode = lib500_types.IO_ERRORTYPE.IO_E_OK) THEN
		eepromBusy:= TRUE;
		IF bRead THEN
			eepromErrorCode := lib500.IO_EEPROM_Read(offset:= uiAddress, length:= wLength, data:= pData);
		ELSE
			eepromErrorCode := lib500.IO_EEPROM_Write(offset:= uiAddress, length:= wLength, data:= pData);
		END_IF
	END_IF
	
ELSIF eepromBusy AND eepromStatus = lib500_types.IO_ERRORTYPE.IO_E_OK THEN
	eepromBusy:= FALSE;
	eepromLoopStep:= eepromLoopStep+1;
	
END_IF
END_METHOD

METHOD PUBLIC initializeEepromEntry
VAR_INPUT
	wAddress: WORD;
	pData: POINTER TO BYTE;
	wSize: WORD;
END_VAR
EEPROM.staAllEntries[iEntryCursor].wAddress:= wAddress;
EEPROM.staAllEntries[iEntryCursor].pData:= pData;
EEPROM.staAllEntries[iEntryCursor].wSize:= wSize;

iEntryCursor:= iEntryCursor+1;
IF (iEntryCursor >= EEPROM.iEepromEntriesCount) THEN
	iEntryCursor:= 0;
END_IF
END_METHOD

END_PROGRAM

// Device/Application/Modules/COMM/Functions/mngCommCan
// This PRG contains non safety-related code.
// The following attribute is autogenerated. Do not remove.
{attribute 'location':='16#800'}
PROGRAM mngCommCan

VAR CONSTANT 
	MAX_LOOP: BYTE:=20;
END_VAR

VAR_INPUT	
	stCanbus: canBus;
END_VAR
VAR	
	init : BOOL := FALSE;
	stReceiveMaks: canReceiveMask;
	
	MISSED_COUNTER: UINT:= 0;
	LOOP_COUNTER: BYTE;
	COMM_TIMER: UINT :=0;
	eError : CL2.ERROR;
	SEND_Error : CL2.ERROR;
	BUSSTATE:CL2.BUSSTATE;

	hCAN_RX : CL2.CAA.HANDLE := CL2.CAA.gc_hINVALID;
		
	hRxMsg : CL2.CAA.HANDLE := CL2.CAA.gc_hINVALID;
	pRxData : POINTER TO CL2.CL2I.DATA;
	ctMsgLeft : CL2.CAA.COUNT;
	
	CAN_RX_COUNT: INT:=0;
	CAN_RX_BUFFER	: ARRAY [0..7] OF BYTE;		
	CAN_TX_BUFFER	: ARRAY [0..7] OF BYTE;		

	CMD_ADDR: UINT:=0;
	CMD_PROG: UINT:=0;
	CMD_DATA: UINT:=0;
	CMD_DNODE: UINT:=0;
	CMD_SNODE: UINT:=0;
	CMD_TYPE: BYTE:=0;
	CMD_FREE: BYTE:=0;
		
	TX_COMM: BOOL:=FALSE;
	
	RSP_ADDR: UINT:=0;
	RSP_PROG: UINT:=0;
	RSP_DATA: UINT:=0;
	RSP_DNODE: UINT:=0;
	RSP_SNODE: UINT:=0;
	RSP_TYPE: BYTE:=0;
	RSP_FREE: BYTE:=0;
	RSP_CONF: ULINT:=0; // variabile temporanea per la compressione 	
END_VAR

VAR
	iTemp1: INT;
	iTemp2: INT;
END_VAR


IF (init = FALSE) THEN	
	mngInit();
ELSE
	LOOP_COUNTER:= MAX_LOOP;
	//VERIFICA STATO BUS
	BUSSTATE:=CL2.GetBusState(stCanbus.stChannel.driver,ADR(eError));
	IF (BUSSTATE = CL2.BUSSTATE.BUSOFF) THEN
		CL2.ResetBusAlarm(stCanbus.stChannel.driver);
	END_IF
	
	// RICEZIONE DEL MESSAGGIO
	catchMessages();
	mngMessage();
	mngResponse();	
	
	//CICLO PER SVUOTARE IL BUFFER DI RICEZIONE
	WHILE ((LOOP_COUNTER > 0) AND (ctMsgLeft > 0)) DO 
		catchMessages();
		mngMessage();
		mngResponse();	
		LOOP_COUNTER:= LOOP_COUNTER-1;
	END_WHILE 

	// ***************** Gestione timer online ***************** //
	
	IF COMM_TIMER>0 THEN
		COMM_TIMER:=COMM_TIMER-1;
		grComm.bCommunicationActive:=TRUE;
	ELSE
		grComm.bCommunicationActive:=FALSE;
	END_IF
END_IF

METHOD PRIVATE mngInit
VAR_INPUT
END_VAR
IF stCanbus.bActive AND stCanbus.stChannel.bInitialized THEN
	registerReceiveMask(udiId:= grComm.uiProtocolMessageID, stCanBus:=stCanbus, receiveMask:= stReceiveMaks);
	init:= stReceiveMaks.bInitialized;
END_IF
END_METHOD

METHOD PRIVATE catchMessages
VAR_INPUT
END_VAR
// ***************** Cattura messaggi ***************** //

IF readMessage(stReceiveMask:=stReceiveMaks, byaReceivedData=> CAN_RX_BUFFER) > 0 THEN
	CAN_RX_COUNT:=CAN_RX_COUNT+1;
END_IF
END_METHOD

METHOD PRIVATE mngMessage
VAR_INPUT
END_VAR

VAR
	CMD_CONF: ULINT:=0; // variabile temporanea per l'estrazione 
	EEPROM_OP_RESULT: BOOL:= FALSE;
	GETSETVAR_OP_RESULT: BOOL:= FALSE;
END_VAR
// ***************** Elaborazione comando ***************** //

IF CAN_RX_COUNT > 0 THEN
	
	CAN_RX_COUNT:= CAN_RX_COUNT-1; 
	
	CMD_ADDR:= CAN_RX_BUFFER[1];
	CMD_ADDR:= SHL(CMD_ADDR, 8) OR CAN_RX_BUFFER[0];
	CMD_DATA:= CAN_RX_BUFFER[3];
	CMD_DATA:= SHL(CMD_DATA,8) OR CAN_RX_BUFFER[2];
		
	CMD_CONF:= CAN_RX_BUFFER[7];
	CMD_CONF:= SHL(CMD_CONF, 8) OR CAN_RX_BUFFER[6];
	CMD_CONF:= SHL(CMD_CONF, 8) OR CAN_RX_BUFFER[5];
	CMD_CONF:= SHL(CMD_CONF, 8) OR CAN_RX_BUFFER[4];
	
	CMD_SNODE:= ULINT_TO_UINT( SHR(CMD_CONF, 0) AND 16#003F );
	CMD_DNODE:= ULINT_TO_UINT( SHR(CMD_CONF, 6) AND 16#003F );
	CMD_PROG:= ULINT_TO_UINT( SHR(CMD_CONF, 12) AND 16#0FFF );
	CMD_FREE:= ULINT_TO_BYTE( SHR(CMD_CONF, 24) AND 16#000F );
	CMD_TYPE:= ULINT_TO_BYTE( SHR(CMD_CONF, 28) AND 16#000F );
	
	//CMD_DATA:= CMD_DATA AND LREAL_TO_UINT(EXPT(2, (CMD_DLEN+1)-1));	// Maschera del campo DATA in base alla lunghezza
		
	

	// Se il messaggio non è per me o non è valido exit
	IF ( (NOT(CMD_SNODE = CMD_DNODE) AND (CMD_DNODE = grComm.uiProtocolVirtualNode)) OR CMD_TYPE = grCommMessageType.HeartRateRequest ) THEN

		COMM_TIMER:= grComm.COMM_TIMER_RLD;
			
		// ____ Preimpostazione della risposta ____ //
		RSP_ADDR:= CMD_ADDR; 
		RSP_DATA:= 0;
		RSP_CONF:= 0;
		RSP_SNODE:= grComm.uiProtocolVirtualNode;
		RSP_DNODE:= CMD_SNODE;
		RSP_PROG:= CMD_PROG;
		RSP_FREE:= 0;
		RSP_TYPE:= INT_TO_BYTE(grCommMessageType.ErrorCode);  // fino a prova contraria
		
	
		// ____ Elaborazione comando ____ //
		CASE BYTE_TO_INT(CMD_TYPE) OF
			
			grCommMessageType.GetVariable:
				getsetVarCallback(VAR_ID:=CMD_ADDR, INPUT_VAL:=0, READ:=FALSE, VAR_RET => RSP_DATA, ESITO_OPERAZIONE=>GETSETVAR_OP_RESULT);
				IF GETSETVAR_OP_RESULT = TRUE THEN
					RSP_TYPE:= INT_TO_BYTE(grCommMessageType.ExitCode);
				END_IF
			
			grCommMessageType.SetVariable:
				getsetVarCallback(VAR_ID:=CMD_ADDR, INPUT_VAL:=CMD_DATA, READ:=TRUE, VAR_RET => RSP_DATA, ESITO_OPERAZIONE=>GETSETVAR_OP_RESULT);
				IF GETSETVAR_OP_RESULT = TRUE THEN
					RSP_TYPE:= INT_TO_BYTE(grCommMessageType.ExitCode);
				END_IF
			
			grCommMessageType.HeartRateRequest:
				RSP_TYPE:= INT_TO_BYTE(grCommMessageType.ExitCode);
			
			grCommMessageType.LoadFromEEPROM:
				readAllFromEEPROMCallback(ESITO_OPERAZIONE=>EEPROM_OP_RESULT);
				IF EEPROM_OP_RESULT = TRUE THEN
					RSP_TYPE:= INT_TO_BYTE(grCommMessageType.ExitCode);
				END_IF
			
			grCommMessageType.WriteToEEPROM:
				writeToEEPROMCallback(IGNORE_FLAG:=FALSE, ESITO_OPERAZIONE=>EEPROM_OP_RESULT);
				IF EEPROM_OP_RESULT = TRUE THEN
					RSP_TYPE:= INT_TO_BYTE(grCommMessageType.ExitCode);
				END_IF
					
			grCommMessageType.WriteAllToEEPROM:
				writeToEEPROMCallback(IGNORE_FLAG:=TRUE, ESITO_OPERAZIONE=>EEPROM_OP_RESULT);
				IF EEPROM_OP_RESULT = TRUE THEN
					RSP_TYPE:= INT_TO_BYTE(grCommMessageType.ExitCode);
				END_IF
					
			grCommMessageType.ApplyVariables:
				applyToRamCallback(ESITO_OPERAZIONE=>EEPROM_OP_RESULT);
				IF EEPROM_OP_RESULT = TRUE THEN
					RSP_TYPE:= INT_TO_BYTE(grCommMessageType.ExitCode);
				END_IF
			
			
			ELSE
				;// PASS
						
		END_CASE
		
		TX_COMM:= TRUE;
		
	ELSE	
		MISSED_COUNTER:=MISSED_COUNTER+1;
	END_IF	
	
	CMD_ADDR:= 0;
	CMD_DATA:= 0;
	CMD_CONF:= 0;
	CMD_SNODE:= 0;
	CMD_DNODE:= 0;
	CMD_PROG:= 0;
	CMD_FREE:= 0;
	CMD_TYPE:= 0;
	
	
END_IF
END_METHOD

METHOD PRIVATE mngResponse
VAR_INPUT
END_VAR

VAR
	TMP_NODE: UINT:= 0;
	stMessage: canMessage;
END_VAR
// ***************** Invio messaggio di risposta ***************** //

IF TX_COMM THEN
	
	// ____ Compressione data ____ //		
	TMP_NODE:= RSP_DNODE;
	TMP_NODE:= SHL(TMP_NODE, 6) OR RSP_SNODE;
	
	RSP_CONF:= (RSP_TYPE AND 16#0F);
	RSP_CONF:= SHL(RSP_CONF, 4) OR (RSP_FREE AND 16#0F);
	RSP_CONF:= SHL(RSP_CONF, 12) OR (RSP_PROG AND 16#0FFF);
	RSP_CONF:= SHL(RSP_CONF, 12) OR (TMP_NODE AND 16#0FFF);
	
	
	
	// ____ Invio messaggio ____ //
	
	CAN_TX_BUFFER[0] := UINT_TO_BYTE(SHR(RSP_ADDR, 0) AND 16#FF);	
	CAN_TX_BUFFER[1] := UINT_TO_BYTE(SHR(RSP_ADDR, 8) AND 16#FF);						
	CAN_TX_BUFFER[2] := UINT_TO_BYTE(SHR(RSP_DATA, 0) AND 16#FF);
	CAN_TX_BUFFER[3] := UINT_TO_BYTE(SHR(RSP_DATA, 8) AND 16#FF);
	CAN_TX_BUFFER[4] := ULINT_TO_BYTE(SHR(RSP_CONF, 0) AND 16#FF);	
	CAN_TX_BUFFER[5] := ULINT_TO_BYTE(SHR(RSP_CONF, 8) AND 16#FF);							
	CAN_TX_BUFFER[6] := ULINT_TO_BYTE(SHR(RSP_CONF, 16) AND 16#FF);	
	CAN_TX_BUFFER[7] := ULINT_TO_BYTE(SHR(RSP_CONF, 24) AND 16#FF);	
	
	stMessage.udiId:= grComm.uiProtocolMessageID;
	stMessage.byLength:= 8;
	stMessage.bExtended:= FALSE;
	stMessage.byaData:= CAN_TX_BUFFER;
	sendMessage(stCanBus:=stCanbus, stMessageToSend:= stMessage, Fault=> );
	
	CAN_TX_BUFFER[0]:= 0;
	CAN_TX_BUFFER[1]:= 0;
	CAN_TX_BUFFER[2]:= 0;
	CAN_TX_BUFFER[3]:= 0;
	CAN_TX_BUFFER[4]:= 0;
	CAN_TX_BUFFER[5]:= 0;
	CAN_TX_BUFFER[6]:= 0;
	CAN_TX_BUFFER[7]:= 0;
	TMP_NODE:= 0;
	RSP_CONF:= 0;	
	TX_COMM:= FALSE;
	
END_IF
END_METHOD

METHOD PRIVATE getsetVarCallback: UINT

VAR_INPUT
	VAR_ID: UINT:= 0;
	INPUT_VAL: UINT:= 0; 
	READ: BOOL; // se == 0 significa GET_VAR, altrimenti SET_VAR
END_VAR


VAR_OUTPUT	
	VAR_RET: UINT:= 0;
	ESITO_OPERAZIONE: BOOL:= FALSE;
END_VAR
ESITO_OPERAZIONE:= TRUE;

IF VAR_ID > 0 AND VAR_ID <= grComm.uiVariablesMaxIndex THEN
	
	IF READ = FALSE AND grComm.staVariables[VAR_ID].accessRights <> grCommAccessRight.NoAccess THEN
		VAR_RET:= grComm.staVariables[VAR_ID].uiValue;
	ELSIF grComm.staVariables[VAR_ID].accessRights = grCommAccessRight.ReadWrite THEN
		IF (INPUT_VAL < grComm.staVariables[VAR_ID].uiLowerValidValue OR INPUT_VAL > grComm.staVariables[VAR_ID].uiHigherValidValue) THEN
			INPUT_VAL:= grComm.staVariables[VAR_ID].uiDefaultValue;
		END_IF
		grComm.staVariables[VAR_ID].uiValue:= INPUT_VAL;
		grComm.staVariables[VAR_ID].status:= grCommVariableStatus.ModifiedByRemote;
	ELSE
		ESITO_OPERAZIONE:= FALSE;
		grComm.staVariables[VAR_ID].status:= grCommVariableStatus.Error;
	END_IF
	
ELSE
	(* Requested ID is invalid *)
	ESITO_OPERAZIONE:= FALSE;
END_IF
END_METHOD

METHOD PRIVATE applyToRamCallback: BOOL;
VAR_INPUT
END_VAR

VAR_OUTPUT
	ESITO_OPERAZIONE: BOOL:= FALSE;
END_VAR
grComm.bTriggerApplyToRAM:= TRUE;
ESITO_OPERAZIONE:= TRUE;
END_METHOD

METHOD PRIVATE readAllFromEEPROMCallback: BOOL;
VAR_INPUT
END_VAR


VAR_OUTPUT
	ESITO_OPERAZIONE: BOOL:= FALSE;
END_VAR

VAR
	uiVarIterator: UINT;
END_VAR
grComm.bTriggerReadFromEEPROM:= TRUE;

ESITO_OPERAZIONE:= TRUE;
END_METHOD

METHOD PRIVATE writeToEEPROMCallback: BOOL;
VAR_INPUT
	IGNORE_FLAG: BOOL:= FALSE;
END_VAR

VAR_OUTPUT
	ESITO_OPERAZIONE: BOOL:= FALSE;
END_VAR
applyToRamCallback();
grComm.bTriggerWriteAllToEEPROM:= (IGNORE_FLAG);
grComm.bTriggerWriteToEEPROM:= (NOT IGNORE_FLAG);

ESITO_OPERAZIONE:= TRUE;
END_METHOD

METHOD PUBLIC applyToRAM
VAR
	uiVarIterator: UINT;
END_VAR
FOR uiVarIterator:= 1 TO grcomm.uiVariablesMaxIndex BY 1 DO
	IF mngCommCan.isVariableValid(grcomm.staVariables[uiVarIterator]) AND grcomm.staVariables[uiVarIterator].status = grCommVariableStatus.ModifiedByRemote THEN
		grcomm.staVariables[uiVarIterator].pointerToSystemVar^:= grcomm.staVariables[uiVarIterator].uiValue;
		grcomm.staVariables[uiVarIterator].status:= grCommVariableStatus.Pristine;
	END_IF
END_FOR
END_METHOD

METHOD PUBLIC isVariableValid : BOOL
VAR_INPUT
	variable: grCommVar;
END_VAR
isVariableValid:= (
	variable.pointerToSystemVar > 0
	);
END_METHOD

METHOD PUBLIC initializeVariable : grCommVar
VAR_INPUT
	pointerToSystemVar: POINTER TO UINT;
	accessRights: grCommAccessRight;
	uiDefaultValue: UINT;
	uiLowerValidValue: UINT;
	uiHigherValidValue: UINT;
END_VAR

VAR 
	newVar: grCommVar;
	tmpVal: UINT;
END_VAR
newVar.pointerToSystemVar:= pointerToSystemVar;
newVar.accessRights:= accessRights;
newVar.uiDefaultValue:= uiDefaultValue;
newVar.uiLowerValidValue:= uiLowerValidValue;
newVar.uiHigherValidValue:= uiHigherValidValue;

tmpVal:= pointerToSystemVar^;
IF(tmpVal < uiLowerValidValue OR tmpVal > uiHigherValidValue) THEN
	tmpVal:= uiDefaultValue;
	pointerToSystemVar^:= uiDefaultValue;
END_IF
newVar.uiValue:= tmpVal;

initializeVariable:= newVar;
END_METHOD

END_PROGRAM

// Device/Application/Modules/Canbus/Functions/registerReceiveMask
// This PRG contains non safety-related code.
// The following attribute is autogenerated. Do not remove.
{attribute 'location':='16#800'}
PROGRAM registerReceiveMask
VAR_INPUT
	stCanBus: canBus;
	udiId: UDINT:= 0;
	udiCobIdMask: UDINT:= 16#1FFFFFFF;
	xExtended: BOOL:= TRUE;
END_VAR
VAR_IN_OUT
	receiveMask: canReceiveMask;
END_VAR

IF (udiId > 0) THEN	
	receiveMask.udiId:= udiId;
	receiveMask.udiCobIdMask:= udiCobIdMask;
	checkReceiveMaskInitialization(stCan:= stCanBus.stChannel, stReceiveMask:= receiveMask);
	receiveMask.bActive:= TRUE;
END_IF

END_PROGRAM

// Device/Application/Modules/Canbus/Functions/checkReceiveMaskInitialization
// This PRG contains non safety-related code.
// The following attribute is autogenerated. Do not remove.
{attribute 'location':='16#800'}
PROGRAM checkReceiveMaskInitialization
VAR_INPUT
	stCan: can;
END_VAR
VAR_IN_OUT
	stReceiveMask: canReceiveMask;
END_VAR
VAR	
	cobIdMask: CL2.CL2I.COBID:= 16#1FFFFFFF; 
	xRTRValue: BOOL:= FALSE;
	xRTRMask: BOOL:= FALSE;
	x29BitIdValue: BOOL:= FALSE; 
	x29BitIdMask: BOOL:= FALSE;
	xTransmitValue: BOOL:= FALSE; 
	xTransmitMask: BOOL:= TRUE;
	xAlwaysNewest: BOOL:= FALSE; 
	eEvent: CL2.CB.EVENT:= 0;
	xEnableSyncWindow: BOOL:= FALSE; 
END_VAR

IF (stCan.bInitialized) AND (stReceiveMask.stCAAMask = CL2.CAA.gc_hINVALID) THEN	
	stReceiveMask.stCAAMask := CL2.CreateMaskReceiver(
		hDriver := stCan.driver, 
		cobIdValue := stReceiveMask.udiId, 
		cobIdMask := stReceiveMask.udiCobIdMask, 
		xRTRValue := xRTRValue, 
		xRTRMask := xRTRMask, 
		x29BitIdValue := x29BitIdValue, 
		x29BitIdMask := x29BitIdMask, 
		xTransmitValue := xTransmitValue, 
		xTransmitMask := xTransmitMask, 
		xAlwaysNewest := xAlwaysNewest, 
		eEvent := eEvent,
		xEnableSyncWindow := xEnableSyncWindow, 
		peError := 0
	);
	
	(*hReceiver := CL2.CreateMaskReceiver(hDriver := canbus.stChannel.driver,
					cobIdValue := 16#18FFFF00, 
					cobIdMask := 16#1F0000FF, 
					xRTRValue := FALSE, //no RTR messages
					xRTRMask := TRUE, //activate RTR filter ==> xRTRValue will be checked
					x29BitIdValue := TRUE, //no 29 bit CAN messages
					x29BitIdMask := TRUE, //activate 29 bit filter ==> x29BitIdValue will be checked
					xTransmitValue := FALSE, //only receive messages, no transmit message loopback
					xTransmitMask := TRUE, //activate transmit mask filter ==> xTransmitValue will be checked
					xAlwaysNewest := FALSE, //FALSE := receiver with queue; TRUE: only newest message
					eEvent := 0, //no receive event
					xEnableSyncWindow := FALSE, //not implemented
					peError := ADR(fault) //optional pointer to error
				);*)
END_IF

IF stReceiveMask.stCAAMask <> CL2.CAA.gc_hINVALID THEN
	stReceiveMask.bInitialized:= TRUE;
END_IF

END_PROGRAM

// Device/Application/Modules/Canbus/Functions/readMessage
// This PRG contains non safety-related code.
// The following attribute is autogenerated. Do not remove.
{attribute 'location':='16#800'}
FUNCTION readMessage: INT;
VAR_IN_OUT
	stReceiveMask: canReceiveMask;
END_VAR
VAR_OUTPUT
	readCount: INT;
	byaReceivedData: ARRAY [0..7] OF BYTE;
END_VAR
VAR	
	iCounter: INT:= 0;
	iReceivedCount: INT:= 0;
	stReceivedMessage: CL2.CAA.HANDLE := CL2.CAA.gc_hINVALID;
	stReceiveError: CL2.ERROR;
	usiTmpData: ARRAY [0..7] OF USINT;
END_VAR

iReceivedCount:= 0;
IF stReceiveMask.bActive THEN
	stReceivedMessage:= CL2.Read(hReceiverId:=stReceiveMask.stCAAMask, pctMsgLeft:=ADR(stReceiveMask.stMessagesLeft), peError:=ADR(stReceiveError));
		
	IF stReceivedMessage <> CL2.CAA.gc_hINVALID THEN
		usiTmpData:= CL2.GetMessageDataPointer(hMessage:=stReceivedMessage, peError:=ADR(stReceiveError))^;
		FOR iCounter:=0 TO 7 BY 1 DO
			byaReceivedData[iCounter]:= USINT_TO_BYTE(usiTmpData[iCounter]);
		END_FOR
		CL2.FreeMessage(hMessage:= stReceivedMessage);
		iReceivedCount:= 1;
	END_IF
END_IF
readCount:= iReceivedCount;

// Per l'uso come function
readMessage:= readCount;

END_FUNCTION

// Device/Application/Modules/Canbus/Functions/sendMessage
// This PRG contains non safety-related code.
// The following attribute is autogenerated. Do not remove.
{attribute 'location':='16#800'}
PROGRAM sendMessage

VAR_INPUT
	stCanBus: canBus;
	stMessageToSend: canMessage;
END_VAR

VAR_OUTPUT
	Fault : CL2.ERROR;
END_VAR

VAR
	stCan: can;
	EXT : BOOL;
	ID : CL2.CL2I.COBID;
	LEN : USINT;
	TX_pointer	: POINTER TO CL2.CL2I.DATA;
	DRIVER : CL2.CAA.HANDLE;
	
	
	hTxMsg : CL2.CAA.HANDLE := CL2.CAA.gc_hINVALID;
	x29Bit : BOOL;
	xRTR : BOOL;
	xTxFrame : BOOL;
	eError : CL2.ERROR;
	pTxData : POINTER TO CL2.CL2I.DATA;
	diMsgRecv: DINT;
	i : INT;
END_VAR

stCan:= stCanBus.stChannel;
EXT:=stMessageToSend.bExtended;
ID:= stMessageToSend.udiId;
LEN:= stMessageToSend.byLength; 
TX_pointer:= ADR(stMessageToSend.byaData); 
DRIVER:= stCan.driver;

checkBusState(stCan:= stCan);		
		
IF(TRUE (*ID > 0*)) THEN		
	IF(LEN > 8) THEN
		LEN:= 8;
	END_IF
	hTxMsg := CL2.CreateMessage(
		hDriver := DRIVER, 
		cobID := ID, 
		usiLength := LEN, 
		xRTR := xRTR, 
		x29BitID := EXT, 
		peError := ADR(eError));
		
	IF hTxMsg <> CL2.CAA.gc_hINVALID THEN
		pTxData := CL2.GetMessageDataPointer(hMessage := hTxMsg, peError := ADR(eError));
		IF pTxData <> CL2.CAA.gc_pNULL AND LEN <> 0 THEN
			FOR i := 0 TO LEN - 1 DO
				pTxData^[i] := TX_pointer^[i];
			END_FOR
		END_IF
		eError := CL2.Write(hDriver := DRIVER, hMessage := hTxMsg, usiPriority := 1, xEnableSyncWindow := FALSE);
		IF eError <> CL2.ERROR.NO_ERROR THEN
			CL2.FreeMessage(hMessage := hTxMsg);
		END_IF
		hTxMsg := CL2.CAA.gc_hINVALID;
		pTxData := CL2.CAA.gc_pNULL;
		Fault:= stCan.transmitError;
	END_IF
END_IF

END_PROGRAM

// Device/Application/Modules/Canbus/Functions/checkBusState
// This PRG contains non safety-related code.
// The following attribute is autogenerated. Do not remove.
{attribute 'location':='16#800'}
PROGRAM checkBusState
VAR_INPUT
	stCan: can;
END_VAR
VAR
	stResetResult: CL2.ERROR:= CL2.ERROR.INVALID_HANDLE;
END_VAR

IF (stCan.bInitialized) AND	(stCan.busStatus <> CL2.BUSSTATE.ERR_FREE) AND (stCan.busStatus <> CL2.BUSSTATE.ACTIVE) THEN
	stResetResult:= CL2.ResetBusAlarm(hDriver:= stCan.driver);
END_IF

END_PROGRAM

// Device/Application/Program logic/Tasks/CanCommunication
PROGRAM CanCommunication
VAR CONSTANT
	uiNode: UINT:= 16#10;
	displayNode: BYTE:= 16#DD;
END_VAR
VAR
	xInitialized: BOOL:= FALSE;
	stCanbusPC: canBus;	
	uiSendVariablesTimerMs: UINT;
	uiStartupTimerMs: UINT:= 60000;
	
	PC_msg_config: canReceiveMask;
	displayMsgIO: canReceiveMask;
	
	uiAntiBumpTimer: UINT:= 0;
	uiAntiBumpIntervalMs: UINT:= 100;
	uiDisplayMsgIOTimerMs: UINT;
	
	byMsgSendStep: BYTE:= 0;
END_VAR

IF NOT xInitialized THEN
	stCanbusPC:= fieldbus.can[1];
	xInitialized:= initialize();
	
ELSE
	IF uiSendVariablesTimerMs = 0 THEN
		uiSendVariablesTimerMs:= 100;
		sendData_to_PC();
	ELSE
		Utils.decrementUINT(uiSendVariablesTimerMs, 10);
	END_IF
	reciveData_from_PC();
	Utils.decrementUINT(uiStartupTimerMs, 10);
END_IF

METHOD PRIVATE sendData_to_PC
VAR
	msg: canMessage;
	rTmpAirPressure: REAL;
	uiTmpSpeed: UINT;
END_VAR
msg.bExtended:= FALSE;

CASE byMsgSendStep OF
	0:
		msg.udiId:= 16#100 ;
		msg.byLength:= 8;
		
		msg.byaData[0].0 := varInput.xInput_1; 
		msg.byaData[0].1 := varInput.xInput_2; 
		msg.byaData[0].2 := varInput.xInput_3; 
		msg.byaData[0].3 := varInput.xInput_4; 
		msg.byaData[0].4 := varInput.xInput_5;  
		msg.byaData[0].5 := varInput.xInput_6;  
		msg.byaData[0].6 := varInput.xInput_7;  
		msg.byaData[0].7 := varInput.xInput_8;  
                           
		msg.byaData[1].0 := varInput.xInput_9;
		msg.byaData[1].1 := varInput.xInput_10;
		msg.byaData[1].2 := varInput.xInput_11;
		msg.byaData[1].3 := varInput.xInput_12;
		msg.byaData[1].4 := varInput.xInput_13;
		msg.byaData[1].5 := varInput.xInput_14;
		msg.byaData[1].6 := varInput.xInput_15;
		msg.byaData[1].7 := varInput.xInput_16;
                          
		msg.byaData[2].0 := varInput.xInput_17; 
		msg.byaData[2].1 := varInput.xInput_18; 
		msg.byaData[2].2 := varInput.xInput_19;
		msg.byaData[2].3 := varInput.xInput_20;
		
		msg.byaData[3] := WORD_TO_BYTE(sysIO.digitalInput.input_122.wCurrent);
		
END_CASE
	
sendMessage(stCanBus:= stCanbusPC, stMessageToSend:= msg);
END_METHOD

METHOD PRIVATE reciveData_from_PC
VAR
	byaData: ARRAY[0..7] OF BYTE;
END_VAR


IF readMessage(stReceiveMask:= PC_msg_config, byaReceivedData=> byaData) > 0 THEN
	varOutput.xOutput_1 := byaData[0].0;
	varOutput.xOutput_2 := byaData[0].1;
	varOutput.xOutput_3 := byaData[0].2;
	varOutput.xOutput_4 := byaData[0].3;
	varOutput.xOutput_5 := byaData[0].4;
	varOutput.xOutput_6 := byaData[0].5;
	varOutput.xOutput_7 := byaData[0].6;
	varOutput.xOutput_8 := byaData[0].7;
	
	varOutput.xOutput_9  := byaData[1].0;
	varOutput.xOutput_10 := byaData[1].1;
	varOutput.xOutput_11 := byaData[1].2;
	varOutput.xOutput_12 := byaData[1].3;
	varOutput.xOutput_13 := byaData[1].4;
	varOutput.xOutput_14 := byaData[1].5;
	varOutput.xOutput_15 := byaData[1].6;
	varOutput.xOutput_16 := byaData[1].7;
	
	varOutput.xOutput_17 := byaData[2].0;
	varOutput.xOutput_18 := byaData[2].1;
	varOutput.xOutput_19 := byaData[2].2;
	varOutput.xOutput_20 := byaData[2].3;
	
	uiDisplayMsgIOTimerMs:= 30000;
END_IF	

Utils.decrementUINT(uiAntiBumpTimer, 10);
Utils.decrementUINT(uiDisplayMsgIOTimerMs, 10);


IF uiDisplayMsgIOTimerMs = 0 THEN
	varOutput.xOutput_1 := FALSE;
	varOutput.xOutput_2 := FALSE;
	varOutput.xOutput_3 := FALSE;
	varOutput.xOutput_4 := FALSE;
	varOutput.xOutput_5 := FALSE;
	varOutput.xOutput_6 := FALSE;
	varOutput.xOutput_7 := FALSE;
	varOutput.xOutput_8 := FALSE;
END_IF
GVL.xDPFRegenerationRequestInput:= display.xInput1;
END_METHOD

METHOD PRIVATE initialize: BOOL;
VAR
	xRet: BOOL;
END_VAR
initialize:= FALSE;
IF stCanbusPC.bActive AND stCanbusPC.stChannel.bInitialized THEN
	registerReceiveMask(udiId:= 16#400, stCanBus:=stCanbusPC, receiveMask:= PC_msg_config);
	
	initialize:= PC_msg_config.bInitialized;
END_IF
END_METHOD

END_PROGRAM

// Device/Application/Modules/Utils/Utils
PROGRAM Utils

VAR CONSTANT
	PWM_ON : WORD :=65000;
	PWM_OFF : WORD :=0;
END_VAR

VAR
	linTrafo: LIN_TRAFO;
END_VAR

METHOD decrementUINT
VAR_IN_OUT
	input: UINT;
END_VAR
VAR_INPUT
	step: UINT;
END_VAR
IF(step > input) THEN 
	input:= 0;
ELSE
	input:= input - step;
END_IF
END_METHOD

METHOD PUBLIC bytesToUInt16 : UINT
VAR_INPUT
	mostSignificantByte: BYTE;
	leastSignificantByte: BYTE;
END_VAR
bytesToUInt16:= SHL(BYTE_TO_UINT(mostSignificantByte), 8) OR leastSignificantByte;
END_METHOD

METHOD PUBLIC toggle
VAR_IN_OUT
	bValue: BOOL;
END_VAR
bValue:= NOT bValue;
END_METHOD

METHOD PUBLIC isNaN: BOOL
VAR_INPUT
	rTest: REAL;
END_VAR
isNaN:= NOT(rTest = rTest);
END_METHOD

METHOD PUBLIC updateValueFiltered : REAL
VAR_INPUT
	rCurrentValue: REAL;
	rNewValue: REAL;
	rFilterConstant: REAL;
END_VAR

VAR
	rFilteredValue: REAL;
END_VAR
rFilteredValue:= (rCurrentValue * rFilterConstant) + (rNewValue * (1 - rFilterConstant));
updateValueFiltered:= rFilteredValue;
END_METHOD

METHOD PUBLIC bytesToInt16 : INT
VAR_INPUT
	mostSignificantByte: BYTE;
	leastSignificantByte: BYTE;
END_VAR
bytesToInt16:= WORD_TO_INT(SHL(BYTE_TO_WORD(mostSignificantByte), 8) OR leastSignificantByte);
END_METHOD

METHOD decrementUDINT
VAR_IN_OUT
	input: UDINT;
END_VAR
VAR_INPUT
	step: UDINT;
END_VAR
IF(step > input) THEN 
	input:= 0;
ELSE
	input:= input - step;
END_IF
END_METHOD

METHOD PUBLIC boolToPWMDutyCycle : WORD
VAR_INPUT
	bEnable: BOOL;
END_VAR
IF bEnable THEN
	boolToPWMDutyCycle:= PWM_ON;
ELSE
	boolToPWMDutyCycle:= PWM_OFF;	
END_IF
END_METHOD

METHOD PUBLIC linearize: REAL
VAR_INPUT
	rIn: REAL;
	rInMin: REAL;
	rInMax: REAL;
	rOutMin: REAL;
	rOutMax: REAL;
END_VAR

VAR_OUTPUT
	xError: BOOL;
END_VAR

VAR
	rOut: REAL;
END_VAR
IF rIn < rInMin THEN rIn:= rInMin; END_IF
IF rIn > rInMax THEN rIn:= rInMax; END_IF

linTrafo(
	IN:= rIn,
	IN_MIN:= rInMin,
	IN_MAX:= rInMax,
	OUT_MIN:= rOutMin,
	OUT_MAX:= rOutMax,
	OUT=> rOut,
	ERROR=> xError
);

linearize:= rOut;
END_METHOD

METHOD PUBLIC bytesToUReal16 : REAL
VAR_INPUT
	mostSignificantByte: BYTE;
	leastSignificantByte: BYTE;
END_VAR
bytesToUReal16:= bytesToUInt16(mostSignificantByte, leastSignificantByte);
END_METHOD

METHOD PUBLIC bytesToUDInt32 : UDINT
VAR_INPUT
	byte0: BYTE;
	byte1: BYTE;
	byte2: BYTE;
	byte3: BYTE;
END_VAR
bytesToUDInt32:= SHL(BYTE_TO_UDINT(byte3), 24) OR SHL(BYTE_TO_UDINT(byte2), 16) OR SHL(BYTE_TO_UDINT(byte1), 8) OR byte0;
END_METHOD

METHOD incrementUINT
VAR_IN_OUT
	input: UINT;
END_VAR
VAR_INPUT
	step: UINT;
END_VAR
IF(step >= (16#FFFF - step)) THEN 
	input:= 16#FFFF;
ELSE
	input:= input + step;
END_IF
END_METHOD

END_PROGRAM

// Device/Application/Program logic/Tasks/MAIN
PROGRAM MAIN
VAR
	xStop: BOOL:= FALSE;
	init : BOOL := FALSE;
	INIT_STEP : UINT:=0;
	result : RTS_IEC_RESULT;
	DeviceName : WSTRING(255) := "";
	DeviceNameLen : UDINT := 255;
	TargetId : DWORD := 0;
	NodeName : WSTRING(255) := "";
	NodeNameLen : UDINT := 255;
	OperatingSystemId : UDINT := 0;
	ProcessorId : UDINT := 0;
	SerialNumber : POINTER TO STRING := 0;
	SerialNumberLen : DINT := 255;
	TargetType : DWORD := 0;
	VendorName : WSTRING(255) := "";
	VendorNameLen : UDINT := 255;
	Version : DWORD := 0;
	
	error_code : lib500_types.IO_ERRORTYPE := lib500_types.IO_ERRORTYPE.IO_E_OK;
		
	shutdownCounterMillis: UDINT:= 30 * 1000;
	uiPowerOnTimeMs: UINT:= 0;
END_VAR

// check, if in init phase
IF (init = FALSE) THEN
	CASE INIT_STEP OF
	0:	
		// SysTargetGetDeviceName()
		result := SysTarget.SysTargetGetDeviceName(
			pwszName:= ADR(DeviceName),
			pnMaxLength:= ADR(DeviceNameLen));
		
		// SysTargetGetId()
		result := SysTarget.SysTargetGetId(
			pulTargetId:= ADR(TargetId));
		
		// SysTargetGetNodeName()
		result := SysTarget.SysTargetGetNodeName(
			pwszName:= ADR(NodeName), 
			pnMaxLength:= ADR(NodeNameLen));
		
		// SysTargetGetOperatingSystemId()
		result := SysTarget.SysTargetGetOperatingSystemId(
			pudiOperatingSystemId:= ADR(OperatingSystemId));
		
		// SysTargetGetProcessorId()
		result := SysTarget.SysTargetGetProcessorId(
			pudiProcessorId:= ADR(ProcessorId));
		
		// SysTargetGetSerialNumber()
		result := SysTarget.SysTargetGetSerialNumber(
			ppsSerialNumber:= ADR(SerialNumber),
			pnMaxLen:= ADR(SerialNumberLen));
		
		// SysTargetGetType()
		result := SysTarget.SysTargetGetType(
			pulType:= ADR(TargetType));
		
		// SysTargetGetVendorName()
		result := SysTarget.SysTargetGetVendorName(
			pwszName:= ADR(VendorName),
			pnMaxLength:= ADR(VendorNameLen));
		
		// SysTargetGetVersion()
		result := SysTarget.SysTargetGetVersion(
			pulVersion:= ADR(Version));
		
		IF DeviceName = "HY-TTC 540" THEN
			GVL.MODELLO_CENTRALINA:= 1;
		ELSIF DeviceName = "HY-TTC 580" THEN
			GVL.MODELLO_CENTRALINA:= 2;
		END_IF								 
		 
		INIT_STEP:=INIT_STEP+1;	
	1:	
		//MNG_RW_EEPROM();
		//IF EEPROM.EEPROM_ST = TRUE THEN
			checkParameters();
			INIT_STEP:=INIT_STEP+1;	
		//END_IF
		
	2:
		IF NOT sysIO.bIOInitialized THEN
			initializeIO();
			IF sysIO.bIOInitialized THEN INIT_STEP:=INIT_STEP+1; END_IF
		END_IF
		
	3:		
		IF NOT fieldbus.bCanbusInitialized THEN
			setupCanbus();
		ELSE
			init:= TRUE;
		END_IF
	END_CASE							  
END_IF

IF (init = TRUE) THEN	
	IF xStop THEN RETURN; END_IF
	checkParameters();
	
	io_module.getInputs();	
	IO.xECUK15:= sysIO.analogInput.ecuK15_p207.dwValue > 10000; 
	
	IF (IO.xECUK15) THEN
		// Esecuzione regolare
		mainLoop();
	ELSIF NOT GVL.xAllowSystemShutdown THEN
		postrun();
	ELSE
		shutdown();
	END_IF
	
	IF uiPowerOnTimeMs < 65000 THEN uiPowerOnTimeMs:= uiPowerOnTimeMs +10; END_IF
	
	UI_PRG();
	io_module.setOutputs();
	system.xFirstCycle:= FALSE;
	
END_IF

METHOD PRIVATE mainLoop
VAR_INPUT
END_VAR
//mngCanbusStatus();	
J1939_PRG();
MachineLogic_PRG();


IF system.xHazardStatus THEN
	shutdownCounterMillis:= 6 * 60 * 60 * 1000; // 6 ore
ELSE
	shutdownCounterMillis:= 30 * 1000;
END_IF

sysIO.digitalOutput.displayK15_p166.bValue:= TRUE;
END_METHOD

ACTION postrun:
Utils.decrementUDINT(shutdownCounterMillis, 10);
GVL.xAllowSystemShutdown:= ((NOT system.xHazardStatus) OR 
							(shutdownCounterMillis = 0)) AND
							uiPowerOnTimeMs > 10000; // devono essere passati almeno 10 secondi dal key-on per poter spegnere (per K15 display)
END_ACTION

ACTION shutdown:

error_code:= lib500.IO_POWER_Set(lib500_types.IO_POWER_CHANNEL.IO_K15, lib500_types.IO_POWER_STATE.IO_POWER_OFF);
END_ACTION

METHOD PRIVATE checkParameters
VAR_INPUT
END_VAR
END_METHOD

ACTION setupCanbus:
IF NOT fieldbus.bCanbusInitialized THEN
	fieldbus.can[0].bActive:= FALSE;
	fieldbus.can[1].bActive:= TRUE; // J1939
	fieldbus.can[2].bActive:= TRUE; // display
	fieldbus.can[3].bActive:= FALSE;
	fieldbus.can[4].bActive:= TRUE; //Modifica Martella
	fieldbus.can[5].bActive:= FALSE;
	fieldbus.can[6].bActive:= FALSE;
	fieldbus.bCanbusInitialized:= initializeCanbus();	
END_IF
END_ACTION

END_PROGRAM

// Device/Application/Modules/IOs/initializeIO
PROGRAM initializeIO
VAR
	bInstantiated: BOOL:= FALSE;
END_VAR

VAR CONSTANT
	TTC_540: BYTE:= 1;
	TTC_580: BYTE:= 2;
END_VAR

IF NOT bInstantiated THEN 
	instantiatePowerStages();
	
	instantiateDigitalInputs();
	instantiateAnalogInputs();
	instantiatePWDInputs();
	
	instantiateDigitalOutputs();
	instantiatePWMOutputs();
	instantiateVoltageOutputs();
	
	bInstantiated:= TRUE;
END_IF

sysIO.bIOInitialized:= io_module.initializeIO(GVL.MODELLO_CENTRALINA);

METHOD PRIVATE instantiateAnalogInputs
VAR_INPUT
END_VAR
io_module.instantiateADC(	
	outPointer:= ADR(sysIO.analogInput.ecuK15_p207), 
	byChannel:= lib500_types.IO_ADC_CHANNEL.IO_ADC_K15, 
	byPullType:= lib500_types.IO_ADC_PUPD.IO_ADC_NO_PULL,
	stADCType:= lib500_types.IO_ADC_TYPE.IO_ADC_ABSOLUTE,
	stADCRange:= lib500_types.IO_ADC_RANGE.IO_ADC_RANGE_32V,
	stADCSensorSupply:= lib500_types.IO_SENSOR_SUPPLY.IO_SENSOR_SUPPLY_0
);
io_module.instantiateADC(	
	outPointer:= ADR(sysIO.analogInput.fuelTankGauge_p103), 
	byChannel:= lib500_types.IO_ADC_CHANNEL.IO_ADC_00, 
	byPullType:= lib500_types.IO_ADC_PUPD.IO_ADC_NO_PULL,
	stADCType:= lib500_types.IO_ADC_TYPE.IO_ADC_RESISTIVE,
	stADCRange:= lib500_types.IO_ADC_RANGE.IO_ADC_NO_RANGE,
	stADCSensorSupply:= lib500_types.IO_SENSOR_SUPPLY.IO_SENSOR_SUPPLY_0
);
io_module.instantiateADC(	
	outPointer:= ADR(sysIO.analogInput.pneumaticTankGauge_p104), 
	byChannel:= lib500_types.IO_ADC_CHANNEL.IO_ADC_02, 
	byPullType:= lib500_types.IO_ADC_PUPD.IO_ADC_NO_PULL,
	stADCType:= lib500_types.IO_ADC_TYPE.IO_ADC_RESISTIVE,
	stADCRange:= lib500_types.IO_ADC_RANGE.IO_ADC_NO_RANGE,
	stADCSensorSupply:= lib500_types.IO_SENSOR_SUPPLY.IO_SENSOR_SUPPLY_0
);
io_module.instantiateADC(	
	outPointer:= ADR(sysIO.analogInput.shiftOilGauge_p128), 
	byChannel:= lib500_types.IO_ADC_CHANNEL.IO_ADC_03, 
	byPullType:= lib500_types.IO_ADC_PUPD.IO_ADC_NO_PULL,
	stADCType:= lib500_types.IO_ADC_TYPE.IO_ADC_RESISTIVE,
	stADCRange:= lib500_types.IO_ADC_RANGE.IO_ADC_NO_RANGE,
	stADCSensorSupply:= lib500_types.IO_SENSOR_SUPPLY.IO_SENSOR_SUPPLY_0
);


io_module.instantiateADC(	
	outPointer:= ADR(sysIO.analogInput.speedLimiterReduction_p251), 
	byChannel:= lib500_types.IO_ADC_CHANNEL.IO_ADC_44, 
	byPullType:= lib500_types.IO_ADC_PUPD.IO_ADC_PD_10K,
	stADCType:= lib500_types.IO_ADC_TYPE.IO_ADC_ABSOLUTE,
	stADCRange:= lib500_types.IO_ADC_RANGE.IO_ADC_RANGE_32V,
	stADCSensorSupply:= lib500_types.IO_SENSOR_SUPPLY.IO_SENSOR_SUPPLY_0
);
END_METHOD

METHOD PRIVATE instantiatePVGOutputs
VAR_INPUT
END_VAR
//io_module.instantiatePVG(			
//	outPointer:= ADR(sysIO.pvgOutput._p161),
//	byChannel:= lib500_types.IO_PWD_CHANNEL.IO_PWD_04,
//	5000
//);
END_METHOD

METHOD PRIVATE instantiateDigitalOutputs
VAR_INPUT
END_VAR
io_module.instantiateDO(				
	outPointer:= ADR(sysIO.digitalOutput.output_149),
	byChannel:= lib500_types.IO_DO_CHANNEL.IO_DO_00		
);
io_module.instantiateDO(				
	outPointer:= ADR(sysIO.digitalOutput.output_150),
	byChannel:= lib500_types.IO_DO_CHANNEL.IO_DO_46
);
io_module.instantiateDO(				
	outPointer:= ADR(sysIO.digitalOutput.output_152),
	byChannel:= lib500_types.IO_DO_CHANNEL.IO_DO_02
);
io_module.instantiateDO(				
	outPointer:= ADR(sysIO.digitalOutput.output_153),
	byChannel:= lib500_types.IO_DO_CHANNEL.IO_DO_16
);
io_module.instantiateDO(				
	outPointer:= ADR(sysIO.digitalOutput.output_154),
	byChannel:= lib500_types.IO_DO_CHANNEL.IO_DO_30
);
io_module.instantiateDO(				
	outPointer:= ADR(sysIO.digitalOutput.output_155),
	byChannel:= lib500_types.IO_DO_CHANNEL.IO_DO_04
);

io_module.instantiateDO(				
	outPointer:= ADR(sysIO.digitalOutput.output_156),
	byChannel:= lib500_types.IO_DO_CHANNEL.IO_DO_18
);
io_module.instantiateDO(				
	outPointer:= ADR(sysIO.digitalOutput.output_157),
	byChannel:= lib500_types.IO_DO_CHANNEL.IO_DO_32
);
io_module.instantiateDO(				
	outPointer:= ADR(sysIO.digitalOutput.output_158),
	byChannel:= lib500_types.IO_DO_CHANNEL.IO_DO_06
);
io_module.instantiateDO(				
	outPointer:= ADR(sysIO.digitalOutput.output_159),
	byChannel:= lib500_types.IO_DO_CHANNEL.IO_DO_20
);
io_module.instantiateDO(				
	outPointer:= ADR(sysIO.digitalOutput.output_173),
	byChannel:= lib500_types.IO_DO_CHANNEL.IO_DO_01
);
io_module.instantiateDO(				
	outPointer:= ADR(sysIO.digitalOutput.output_174),
	byChannel:= lib500_types.IO_DO_CHANNEL.IO_DO_47
);
io_module.instantiateDO(				
	outPointer:= ADR(sysIO.digitalOutput.output_176),
	byChannel:= lib500_types.IO_DO_CHANNEL.IO_DO_03
);
io_module.instantiateDO(				
	outPointer:= ADR(sysIO.digitalOutput.output_177),
	byChannel:= lib500_types.IO_DO_CHANNEL.IO_DO_17
);
io_module.instantiateDO(				
	outPointer:= ADR(sysIO.digitalOutput.output_178),
	byChannel:= lib500_types.IO_DO_CHANNEL.IO_DO_31	
);
io_module.instantiateDO(				
	outPointer:= ADR(sysIO.digitalOutput.output_179),
	byChannel:= lib500_types.IO_DO_CHANNEL.IO_DO_05
);
io_module.instantiateDO(				
	outPointer:= ADR(sysIO.digitalOutput.output_180),
	byChannel:= lib500_types.IO_DO_CHANNEL.IO_DO_19
);
io_module.instantiateDO(				
	outPointer:= ADR(sysIO.digitalOutput.output_181),
	byChannel:= lib500_types.IO_DO_CHANNEL.IO_DO_33
);
io_module.instantiateDO(				
	outPointer:= ADR(sysIO.digitalOutput.output_182),
	byChannel:= lib500_types.IO_DO_CHANNEL.IO_DO_07
);
io_module.instantiateDO(				
	outPointer:= ADR(sysIO.digitalOutput.output_183),
	byChannel:= lib500_types.IO_DO_CHANNEL.IO_DO_21
);
END_METHOD

METHOD PRIVATE instantiateVoltageOutputs
VAR_INPUT
END_VAR
(*io_module.instantiateVOUT(			
	outPointer:= ADR(sysIO.voltageOutput.coolerPumpDrive_p161),
	byChannel:= lib500_types.IO_VOUT_CHANNEL.IO_VOUT_00
);
*)
END_METHOD

METHOD PRIVATE instantiatePWDInputs
VAR_INPUT
END_VAR
(*
io_module.instantiatePWD(			
	outPointer:= ADR(sysIO.pwdInput.speedSensor_p115),
	byChannel:= lib500_types.IO_PWD_CHANNEL.IO_PWD_00,
	pwdMode:= lib500_types.IO_PWD_INC_MODE.IO_PWD_INC_2_COUNT,
	byPullType:= lib500_types.IO_PWD_PUPD.IO_PWD_PU_10K,
	readMode:= pwdReadMode.complex,
	wCountInit:= 32767
);
sysIO.pwdInput.speedSensor_p115.pulseMode:= lib500_types.IO_PWD_PULSE_MODE.IO_PWD_HIGH_TIME;
sysIO.pwdInput.speedSensor_p115.freqMode:= lib500_types.IO_PWD_FREQ_MODE.IO_PWD_FALLING_VAR;
*)

io_module.instantiatePWD(			
	outPointer:= ADR(sysIO.pwdInput.transmissionShaftSensor5000_p175),
	byChannel:= lib500_types.IO_PWD_CHANNEL.IO_PWD_19,
	pwdMode:= lib500_types.IO_PWD_INC_MODE.IO_PWD_INC_2_COUNT,
	byPullType:= lib500_types.IO_PWD_PUPD.IO_PWD_PU_10K,
	readMode:= pwdReadMode.complex,
	wCountInit:= 32767
);
sysIO.pwdInput.transmissionShaftSensor5000_p175.pulseMode:= lib500_types.IO_PWD_PULSE_MODE.IO_PWD_HIGH_TIME;
sysIO.pwdInput.transmissionShaftSensor5000_p175.freqMode:= lib500_types.IO_PWD_FREQ_MODE.IO_PWD_FALLING_VAR;


io_module.instantiatePWD(			
	outPointer:= ADR(sysIO.pwdInput.transmissionShaftSensor7500_p151),
	byChannel:= lib500_types.IO_PWD_CHANNEL.IO_PWD_18,
	pwdMode:= lib500_types.IO_PWD_INC_MODE.IO_PWD_INC_2_COUNT,
	byPullType:= lib500_types.IO_PWD_PUPD.IO_PWD_PD_10K,
	readMode:= pwdReadMode.complex,
	wCountInit:= 32767
);
sysIO.pwdInput.transmissionShaftSensor7500_p151.pulseMode:= lib500_types.IO_PWD_PULSE_MODE.IO_PWD_HIGH_TIME;
sysIO.pwdInput.transmissionShaftSensor7500_p151.freqMode:= lib500_types.IO_PWD_FREQ_MODE.IO_PWD_FALLING_VAR;
sysIO.pwdInput.transmissionShaftSensor7500_p151.byCaptureCount:= 1;
END_METHOD

METHOD PRIVATE instantiatePowerStages
VAR_INPUT
END_VAR
io_module.instantiatePower(			
	outPointer:= ADR(sysIO.powerStage.safetySwitch0),
	byChannel:= lib500_types.IO_POWER_CHANNEL.IO_INT_SAFETY_SW_0,
	mode:= lib500_types.IO_POWER_STATE.IO_POWER_ON
);
														
io_module.instantiatePower(			
	outPointer:= ADR(sysIO.powerStage.safetySwitch1),
	byChannel:= lib500_types.IO_POWER_CHANNEL.IO_INT_SAFETY_SW_1,
	mode:= lib500_types.IO_POWER_STATE.IO_POWER_ON
);
														
io_module.instantiatePower(			
	outPointer:= ADR(sysIO.powerStage.safetySwitch2),
	byChannel:= lib500_types.IO_POWER_CHANNEL.IO_INT_SAFETY_SW_2,
	mode:= lib500_types.IO_POWER_STATE.IO_POWER_ON
);
sysIO.powerStage.safetySwitch2.byMinTTCModel:= TTC_580;

														
io_module.instantiatePower(				
	outPointer:= ADR(sysIO.powerStage.powerStage),
	byChannel:= lib500_types.IO_POWER_CHANNEL.IO_INT_POWERSTAGE_ENABLE,
	mode:= lib500_types.IO_POWER_STATE.IO_POWER_ON
);
														
io_module.instantiatePower(			
	outPointer:= ADR(sysIO.powerStage.sensorSupply0),
	byChannel:= lib500_types.IO_POWER_CHANNEL.IO_SENSOR_SUPPLY_0,
	mode:= lib500_types.IO_POWER_STATE.IO_POWER_ON
);
														
io_module.instantiatePower(			
	outPointer:= ADR(sysIO.powerStage.sensorSupply1),
	byChannel:= lib500_types.IO_POWER_CHANNEL.IO_SENSOR_SUPPLY_1,
	mode:= lib500_types.IO_POWER_STATE.IO_POWER_ON
);
														
io_module.instantiatePower(			
	outPointer:= ADR(sysIO.powerStage.sensorSupply2),
	byChannel:= lib500_types.IO_POWER_CHANNEL.IO_SENSOR_SUPPLY_2,
	mode:= lib500_types.IO_POWER_STATE.IO_POWER_ON_10V
);
END_METHOD

METHOD PRIVATE instantiatePWMOutputs
io_module.instantiatePWM(
	outPointer:= ADR(sysIO.pwmOutput.hazardBtnBacklight_p190),
	byChannel:= lib500_types.IO_PWM_CHANNEL.IO_PWM_22,
	wFrequency:= 100,	
	bPolarity:= TRUE,
	bDiagMargin:= FALSE
);
io_module.instantiatePWM(
	outPointer:= ADR(sysIO.pwmOutput.turtleBtnBacklight_p168),
	byChannel:= lib500_types.IO_PWM_CHANNEL.IO_PWM_11,
	wFrequency:= 100,	
	bPolarity:= TRUE,
	bDiagMargin:= FALSE
);
END_METHOD

METHOD PRIVATE instantiateDigitalInputs
VAR_INPUT
END_VAR
io_module.instantiateDI(				
	outPointer:= ADR(sysIO.digitalInput.input_115),
	byChannel:= lib500_types.IO_DI_CHANNEL.IO_DI_36, 
	byPullType:= lib500_types.IO_DI_PUPD.IO_DI_PD_10K
);
io_module.instantiateDI(				
	outPointer:= ADR(sysIO.digitalInput.input_116),
	byChannel:= lib500_types.IO_DI_CHANNEL.IO_DI_38, 
	byPullType:= lib500_types.IO_DI_PUPD.IO_DI_PD_10K
);
io_module.instantiateDI(				
	outPointer:= ADR(sysIO.digitalInput.input_117),
	byChannel:= lib500_types.IO_DI_CHANNEL.IO_DI_40, 
	byPullType:= lib500_types.IO_DI_PUPD.IO_DI_PD_10K
);
io_module.instantiateDI(				
	outPointer:= ADR(sysIO.digitalInput.input_122),
	byChannel:= lib500_types.IO_DI_CHANNEL.IO_DI_42, 
	byPullType:= lib500_types.IO_DI_PUPD.IO_DI_PD_10K
);
io_module.instantiateDI(				
	outPointer:= ADR(sysIO.digitalInput.input_123),
	byChannel:= lib500_types.IO_DI_CHANNEL.IO_DI_44, 
	byPullType:= lib500_types.IO_DI_PUPD.IO_DI_PD_10K
);
io_module.instantiateDI(				
	outPointer:= ADR(sysIO.digitalInput.input_124),
	byChannel:= lib500_types.IO_DI_CHANNEL.IO_DI_46, 
	byPullType:= lib500_types.IO_DI_PUPD.IO_DI_PD_10K
);
io_module.instantiateDI(				
	outPointer:= ADR(sysIO.digitalInput.input_139),
	byChannel:= lib500_types.IO_DI_CHANNEL.IO_DI_37, 
	byPullType:= lib500_types.IO_DI_PUPD.IO_DI_PD_10K
);
io_module.instantiateDI(				
	outPointer:= ADR(sysIO.digitalInput.input_140),
	byChannel:= lib500_types.IO_DI_CHANNEL.IO_DI_39, 
	byPullType:= lib500_types.IO_DI_PUPD.IO_DI_PD_10K
);
io_module.instantiateDI(				
	outPointer:= ADR(sysIO.digitalInput.input_141),
	byChannel:= lib500_types.IO_DI_CHANNEL.IO_DI_41, 
	byPullType:= lib500_types.IO_DI_PUPD.IO_DI_PD_10K
);
io_module.instantiateDI(				
	outPointer:= ADR(sysIO.digitalInput.input_146),
	byChannel:= lib500_types.IO_DI_CHANNEL.IO_DI_43, 
	byPullType:= lib500_types.IO_DI_PUPD.IO_DI_PD_10K
);
io_module.instantiateDI(				
	outPointer:= ADR(sysIO.digitalInput.input_147),
	byChannel:= lib500_types.IO_DI_CHANNEL.IO_DI_45, 
	byPullType:= lib500_types.IO_DI_PUPD.IO_DI_PD_10K
);
io_module.instantiateDI(				
	outPointer:= ADR(sysIO.digitalInput.input_148),
	byChannel:= lib500_types.IO_DI_CHANNEL.IO_DI_47, 
	byPullType:= lib500_types.IO_DI_PUPD.IO_DI_PD_10K
);
io_module.instantiateDI(				
	outPointer:= ADR(sysIO.digitalInput.input_161),
	byChannel:= lib500_types.IO_DI_CHANNEL.IO_DI_88, 
	byPullType:= lib500_types.IO_DI_PUPD.IO_DI_PD_10K
);
io_module.instantiateDI(				
	outPointer:= ADR(sysIO.digitalInput.input_164),
	byChannel:= lib500_types.IO_DI_CHANNEL.IO_DI_91, 
	byPullType:= lib500_types.IO_DI_PUPD.IO_DI_PD_10K
);
io_module.instantiateDI(				
	outPointer:= ADR(sysIO.digitalInput.input_167),
	byChannel:= lib500_types.IO_DI_CHANNEL.IO_DI_93, 
	byPullType:= lib500_types.IO_DI_PUPD.IO_DI_PD_10K
);
io_module.instantiateDI(				
	outPointer:= ADR(sysIO.digitalInput.input_170),
	byChannel:= lib500_types.IO_DI_CHANNEL.IO_DI_95, 
	byPullType:= lib500_types.IO_DI_PUPD.IO_DI_PD_10K
);
io_module.instantiateDI(				
	outPointer:= ADR(sysIO.digitalInput.input_185),
	byChannel:= lib500_types.IO_DI_CHANNEL.IO_DI_89, 
	byPullType:= lib500_types.IO_DI_PUPD.IO_DI_PD_10K
);
io_module.instantiateDI(				
	outPointer:= ADR(sysIO.digitalInput.input_188),
	byChannel:= lib500_types.IO_DI_CHANNEL.IO_DI_90, 
	byPullType:= lib500_types.IO_DI_PUPD.IO_DI_PD_10K
);
io_module.instantiateDI(				
	outPointer:= ADR(sysIO.digitalInput.input_191),
	byChannel:= lib500_types.IO_DI_CHANNEL.IO_DI_92, 
	byPullType:= lib500_types.IO_DI_PUPD.IO_DI_PD_10K
);
io_module.instantiateDI(				
	outPointer:= ADR(sysIO.digitalInput.input_194),
	byChannel:= lib500_types.IO_DI_CHANNEL.IO_DI_94, 
	byPullType:= lib500_types.IO_DI_PUPD.IO_DI_PD_10K
);
END_METHOD

END_PROGRAM

// Device/Application/Modules/IOs/Functions/io_module
PROGRAM io_module
VAR CONSTANT
	DI_maxIndex: 	INT:= 72;
	ADC_maxIndex: 	INT:= 60;
	DO_maxIndex: 	INT:= 40;
	Power_maxIndex: INT:= 10;
	PWM_maxIndex: 	INT:= 36;
	PWD_maxIndex: 	INT:= 19;
	PVG_maxIndex: 	INT:= 7;
	VOUT_maxIndex: 	INT:= 7;
END_VAR
VAR 
	paAllDigitalInputs:  ARRAY[0..DI_maxIndex] 		OF POINTER TO pinDIO;
	paAllADCInputs: 	 ARRAY[0..ADC_maxIndex] 	OF POINTER TO pinADC;		
	paAllDigitalOutputs: ARRAY[0..DO_maxIndex] 		OF POINTER TO pinDIO;
	paAllPowerOutputs: 	 ARRAY[0..Power_maxIndex] 	OF POINTER TO pinPower;
	paAllPWMOutputs:	 ARRAY[0..PWM_maxIndex] 	OF POINTER TO pinPWM;
	paAllPWDInputs:		 ARRAY[0..PWD_maxIndex]		OF POINTER TO pinPWD;
	paAllPVGOutputs:	 ARRAY[0..PVG_maxIndex] 	OF POINTER TO pinPVG;
	paAllVOUTOutputs:	 ARRAY[0..VOUT_maxIndex] 	OF POINTER TO pinVOUT;
	
	iAllDICursor: 	 INT:= 0;
	iAllADCCursor: 	 INT:= 0;	
	iAllDOCursor: 	 INT:= 0;
	iAllPowerCursor: INT:= 0;
	iAllPWMCursor: 	 INT:= 0;
	iAllPWDCursor: 	 INT:= 0;
	iAllPVGCursor: 	 INT:= 0;
	iAllVOUTCursor:	 INT:= 0;
	
	inputPinError: lib500_types.IO_ERRORTYPE;
	outputPinError: lib500_types.IO_ERRORTYPE;
	initializePinError: lib500_types.IO_ERRORTYPE;
	
	byTTCModel: BYTE:= 0;
END_VAR

METHOD PUBLIC instantiateDI: BOOL;
VAR_INPUT
	outPointer: POINTER TO pinDIO;
	byChannel: BYTE;
	byPullType: BYTE:= 0;
END_VAR
instantiateDIO(outPointer, byChannel, byPullType);

paAllDigitalInputs[iAllDICursor]:= outPointer;
iAllDICursor:= iAllDICursor + 1;

IF iAllDICursor >= DI_maxIndex THEN
	iAllDICursor:= 0;
END_IF
END_METHOD

METHOD PUBLIC instantiatePWM
VAR_INPUT
	outPointer: POINTER TO pinPWM;
	byChannel: BYTE;
	wFrequency: WORD;
	bPolarity: BOOL;
	bDiagMargin: BOOL;
END_VAR
outPointer^.byChannel:= byChannel;
outPointer^.wFrequency:= wFrequency;
outPointer^.bPolarity:= bPolarity;
outPointer^.bDiagMargin:= bDiagMargin;

paAllPWMOutputs[iAllPWMCursor]:= outPointer;
iAllPWMCursor:= iAllPWMCursor + 1;

IF iAllPWMCursor >= PWM_maxIndex THEN
	iAllPWMCursor:= 0;
END_IF
END_METHOD

METHOD PUBLIC instantiatePower
VAR_INPUT
	outPointer: POINTER TO pinPower;
	byChannel: BYTE;
	mode: lib500_types.IO_POWER_STATE;
END_VAR
VAR
	pin: pinPower;
END_VAR
outPointer^.byChannel:= byChannel;
outPointer^.mode:= mode;

paAllPowerOutputs[iAllPowerCursor]:= outPointer;
iAllPowerCursor:= iAllPowerCursor + 1;

IF iAllPowerCursor >= Power_maxIndex THEN
	iAllPowerCursor:= 0;
END_IF
END_METHOD

METHOD PUBLIC instantiateVOUT
VAR_INPUT
	outPointer: POINTER TO pinVOUT;
	byChannel: BYTE;
END_VAR
outPointer^.byChannel:= byChannel;

paAllVOUTOutputs[iAllVOUTCursor]:= outPointer;
iAllVOUTCursor:= iAllVOUTCursor + 1;

IF iAllVOUTCursor >= VOUT_maxIndex THEN
	iAllVOUTCursor:= 0;
END_IF
END_METHOD

METHOD PUBLIC instantiateADC
VAR_INPUT
	outPointer: POINTER TO pinADC;
	byChannel: BYTE;
	byPullType: BYTE;
	stADCType: lib500_types.IO_ADC_TYPE;
	stADCRange: lib500_types.IO_ADC_RANGE;
	stADCSensorSupply: lib500_types.IO_SENSOR_SUPPLY;
END_VAR
outPointer^.byChannel:= byChannel;
outPointer^.byPullType:= byPullType;
outPointer^.stADCType:= stADCType;
outPointer^.stADCRange:= stADCRange;
outPointer^.stADCSensorSupply:= stADCSensorSupply;

paAllADCInputs[iAllADCCursor]:= outPointer;
iAllADCCursor:= iAllADCCursor + 1;

IF iAllADCCursor >= ADC_maxIndex THEN
	iAllADCCursor:= 0;
END_IF
END_METHOD

METHOD getInputs : BOOL
VAR
	iDIIterator: INT;
	iADCIterator: INT;
	iPWDIterator: INT;
	pinDITemp: pinDIO;
	pinADCTemp: pinADC;
	pinPWDTemp: pinPWD;
END_VAR
getInputs:= TRUE;
inputPinError:= lib500_types.IO_ERRORTYPE.IO_E_OK;

FOR iDIIterator:= 0 TO iAllDICursor - 1 BY 1 DO
	IF paAllDigitalInputs[iDIIterator] = 0 THEN CONTINUE; END_IF
	IF NOT paAllDigitalInputs[iDIIterator]^.bInitialized THEN CONTINUE; END_IF
	
	pinDITemp:= paAllDigitalInputs[iDIIterator]^;
	IF pinDITemp.byMinTTCModel > byTTCModel THEN CONTINUE; END_IF
	pinDITemp.stError:= lib500.IO_DI_Get(di_channel:= pinDITemp.byChannel, di_value:= ADR(pinDITemp.bValue));	
	
	(* if pin is a negative input negates bValue so that user code can read TRUE if input is active*)
	IF (pinDITemp.byPullType = lib500_types.IO_DI_PUPD.IO_DI_PU_10K) THEN
		pinDITemp.bValue:= NOT(pinDITemp.bValue);
	END_IF
	
	IF (pinDITemp.stError <> lib500_types.IO_ERRORTYPE.IO_E_OK) THEN
		pinDITemp.bValue:= FALSE;
		getInputs:= FALSE;
		inputPinError:= pinDITemp.stError;
	END_IF
	
	paAllDigitalInputs[iDIIterator]^:= pinDITemp;
	
END_FOR



FOR iADCIterator:= 0 TO iAllADCCursor - 1 BY 1 DO
	IF paAllADCInputs[iADCIterator] = 0 THEN CONTINUE; END_IF
	IF NOT paAllADCInputs[iADCIterator]^.bInitialized THEN CONTINUE; END_IF
	
	pinADCTemp:= paAllADCInputs[iADCIterator]^;
	IF pinADCTemp.byMinTTCModel > byTTCModel THEN CONTINUE; END_IF
	pinADCTemp.stError:= lib500.IO_ADC_Get(adc_channel:= pinADCTemp.byChannel, 
											adc_value:= ADR(pinADCTemp.dwValue), 
											fresh:= ADR(pinADCTemp.bValueFresh));
											
	IF pinADCTemp.stError = lib500_types.IO_ERRORTYPE.IO_E_FET_PROT_REENABLE THEN
		lib500.IO_ADC_ResetProtection(adc_channel:= pinADCTemp.byChannel, ADR(pinADCTemp.byResetCount));
	END_IF
	
	IF (pinADCTemp.stError <> lib500_types.IO_ERRORTYPE.IO_E_OK) THEN
		getInputs:= FALSE;
		inputPinError:= pinADCTemp.stError;
	END_IF
	
	paAllADCInputs[iADCIterator]^:= pinADCTemp;
	
END_FOR



FOR iPWDIterator:= 0 TO iAllPWDCursor - 1 BY 1 DO
	IF paAllPWDInputs[iPWDIterator] = 0 THEN CONTINUE; END_IF
	IF NOT paAllPWDInputs[iPWDIterator]^.bInitialized THEN CONTINUE; END_IF
	
	pinPWDTemp:= paAllPWDInputs[iPWDIterator]^;
	IF pinPWDTemp.byMinTTCModel > byTTCModel THEN CONTINUE; END_IF
	pinPWDTemp.stGetVoltageError:= lib500.IO_PWD_GetVoltage(
		pwd_channel:= pinPWDTemp.byChannel,
		voltage:= ADR(pinPWDTemp.uiVoltage),
		fresh:= ADR(pinPWDTemp.bVoltageFresh)
	);
	
	IF pinPWDTemp.bSetIncrementCount THEN
		pinPWDTemp.bSetIncrementCount:= FALSE;
		pinPWDTemp.stIncSetError := lib500.IO_PWD_IncSet(pinPWDTemp.byChannel, pinPWDTemp.wCountZero);
	END_IF
	
	IF pinPWDTemp.readMode = pwdReadMode.incremental THEN 
		pinPWDTemp.stError:= lib500.IO_PWD_IncGet(
								pinPWDTemp.byChannel,
								ADR(pinPWDTemp.wCount),
								ADR(pinPWDTemp.bChannelA),
								ADR(pinPWDTemp.bChannelB)
							);
							
	ELSIF pinPWDTemp.readMode = pwdReadMode.complex THEN 
		pinPWDTemp.stError:= lib500.IO_PWD_ComplexGet(
								timer_channel:= pinPWDTemp.byChannel,
								frequency:= ADR(pinPWDTemp.dwFrequencyHz),
								pulse_width:= ADR(pinPWDTemp.dwPulseWidth),
								pin_value:= ADR(pinPWDTemp.bChannelA),
								pulse_samples:= ADR(pinPWDTemp.pulseSamples)
							);
							
	END_IF	
											
	IF pinPWDTemp.stError = lib500_types.IO_ERRORTYPE.IO_E_FET_PROT_REENABLE THEN
		lib500.IO_PWD_ResetProtection(pwd_channel:= pinPWDTemp.byChannel, ADR(pinPWDTemp.byResetCount));
	END_IF
	
	IF (pinPWDTemp.stError <> lib500_types.IO_ERRORTYPE.IO_E_OK) THEN
		getInputs:= FALSE;
		inputPinError:= pinPWDTemp.stError;
	END_IF
	
	paAllPWDInputs[iPWDIterator]^:= pinPWDTemp;
	
END_FOR
END_METHOD

METHOD PUBLIC instantiatePWD
VAR_INPUT
	outPointer: POINTER TO pinPWD;
	byChannel: BYTE;
	pwdMode: lib500_types.IO_PWD_INC_MODE;
	wCountInit: WORD;
	byPullType: BYTE:= 0;
	readMode: pwdReadMode;
END_VAR
outPointer^.byChannel:= byChannel;
outPointer^.pwdMode:= pwdMode;
outPointer^.wCountInit:= wCountInit;
outPointer^.byPullType:= byPullType;
outPointer^.readMode:= readMode;

paAllPWDInputs[iAllPWDCursor]:= outPointer;
iAllPWDCursor:= iAllPWDCursor + 1;

IF iAllPWDCursor >= PWD_maxIndex THEN
	iAllPWDCursor:= 0;
END_IF
END_METHOD

METHOD PUBLIC initializeIO: BOOL
VAR_INPUT
	TTCModel: BYTE;
END_VAR
VAR
	iDIIterator: INT;
	iDIOterator: INT;
	iADCIterator: INT;
	iPowerChannelIterator: INT;
	iPWMIterator: INT;
	iPWDIterator: INT;
	iPVGIterator: INT;
	iVOUTIterator: INT;
	
	pinDITemp: pinDIO;
	pinDOTemp: pinDIO;
	pinADCTemp: pinADC;
	pinPCTemp: pinPower;
	pinPWMTemp: pinPWM;
	pinPWDTemp: pinPWD;
	pinPVGTemp: pinPVG;
	pinVOUTTemp: pinVOUT;
END_VAR
initializeIO:= TRUE;
initializePinError:= lib500_types.IO_ERRORTYPE.IO_E_OK;
byTTCModel:= TTCModel;


FOR iPowerChannelIterator:= 0 TO iAllPowerCursor - 1 BY 1 DO
	IF paAllPowerOutputs[iPowerChannelIterator] = 0 THEN CONTINUE; END_IF
	pinPCTemp:= paAllPowerOutputs[iPowerChannelIterator]^;
	IF pinPCTemp.bInitialized OR pinPCTemp.byMinTTCModel > byTTCModel THEN CONTINUE; END_IF
	
	pinPCTemp.stInitError:= lib500.IO_POWER_Set(pin:= pinPCTemp.byChannel, mode:= pinPCTemp.mode);										
	pinPCTemp.bInitialized:= (pinPCTemp.stInitError = lib500_types.IO_ERRORTYPE.IO_E_OK);
	IF(pinPCTemp.stInitError <> lib500_types.IO_ERRORTYPE.IO_E_OK) THEN initializePinError:= pinPCTemp.stInitError; END_IF
	IF NOT pinPCTemp.bInitialized THEN initializeIO:= FALSE; END_IF
	
	paAllPowerOutputs[iPowerChannelIterator]^:= pinPCTemp;
	
END_FOR

(* Inputs *)
FOR iADCIterator:= 0 TO iAllADCCursor - 1 BY 1 DO
	IF paAllADCInputs[iADCIterator] = 0 THEN CONTINUE; END_IF
	pinADCTemp:= paAllADCInputs[iADCIterator]^;
	IF pinADCTemp.bInitialized OR pinADCTemp.byMinTTCModel > byTTCModel THEN CONTINUE; END_IF
	
	pinADCTemp.stInitError:= lib500.IO_ADC_ChannelInit(adc_channel:= pinADCTemp.byChannel, 
														pupd:= pinADCTemp.byPullType,
														adc_type:= pinADCTemp.stADCType,
														range:= pinADCTemp.stADCRange,
														sensor_supply:= pinADCTemp.stADCSensorSupply,
														safety_conf:= 0);					
	
	// per qualche motivo K15 init da errore, ma poi funziona la lettura comunque...
	IF pinADCTemp.byChannel = lib500_types.IO_ADC_CHANNEL.IO_ADC_K15 AND pinADCTemp.stInitError = lib500_types.IO_ERRORTYPE.IO_E_CHANNEL_BUSY THEN
		pinADCTemp.stInitError:= lib500_types.IO_ERRORTYPE.IO_E_OK;
	END_IF
	
	IF (pinADCTemp.stInitError <> lib500_types.IO_ERRORTYPE.IO_E_OK) THEN initializePinError:= pinADCTemp.stInitError; END_IF				
	pinADCTemp.bInitialized:= (pinADCTemp.stInitError = lib500_types.IO_ERRORTYPE.IO_E_OK);	
	IF NOT pinADCTemp.bInitialized THEN initializeIO:= FALSE; END_IF
	
	paAllADCInputs[iADCIterator]^:= pinADCTemp;
	
END_FOR

FOR iDIIterator:= 0 TO iAllDICursor - 1 BY 1 DO
	IF paAllDigitalInputs[iDIIterator] = 0 THEN CONTINUE; END_IF
	pinDITemp:= paAllDigitalInputs[iDIIterator]^;
	IF pinDITemp.bInitialized OR pinDITemp.byMinTTCModel > byTTCModel THEN CONTINUE; END_IF
	
	pinDITemp.stInitError:= lib500.IO_DI_Init(di_channel:= pinDITemp.byChannel, pupd:= pinDITemp.byPullType, limits:= 0);		
	IF(pinDITemp.stInitError <> lib500_types.IO_ERRORTYPE.IO_E_OK) THEN initializePinError:= pinDITemp.stInitError; END_IF								
	pinDITemp.bInitialized:= (pinDITemp.stInitError = lib500_types.IO_ERRORTYPE.IO_E_OK);		
	IF NOT pinDITemp.bInitialized THEN	initializeIO:= FALSE; END_IF
	
	paAllDigitalInputs[iDIIterator]^:= pinDITemp;
	
END_FOR




(* Outputs *)

FOR iDIOterator:= 0 TO iAllDOCursor - 1 BY 1 DO
	IF paAllDigitalOutputs[iDIOterator] = 0 THEN CONTINUE; END_IF
	pinDOTemp:= paAllDigitalOutputs[iDIOterator]^;
	IF pinDOTemp.bInitialized OR pinDOTemp.byMinTTCModel > byTTCModel THEN CONTINUE; END_IF
	
	pinDOTemp.stInitError:= lib500.IO_DO_Init(do_channel:= pinDOTemp.byChannel, diagnostic:= 0,	safety_conf:= 0);	
	IF(pinDOTemp.stInitError <> lib500_types.IO_ERRORTYPE.IO_E_OK) THEN initializePinError:= pinDOTemp.stInitError; END_IF												
	pinDOTemp.bInitialized:= (pinDOTemp.stInitError = lib500_types.IO_ERRORTYPE.IO_E_OK);		
	IF NOT pinDOTemp.bInitialized THEN initializeIO:= FALSE; END_IF
	
	paAllDigitalOutputs[iDIOterator]^:= pinDOTemp;
	
END_FOR



FOR iPWMIterator:= 0 TO iAllPWMCursor - 1 BY 1 DO
	IF paAllPWMOutputs[iPWMIterator] = 0 THEN CONTINUE; END_IF
	pinPWMTemp:= paAllPWMOutputs[iPWMIterator]^;
	IF pinPWMTemp.bInitialized OR pinPWMTemp.byMinTTCModel > byTTCModel THEN CONTINUE; END_IF
	
	pinPWMTemp.stInitError:= lib500.IO_PWM_Init(pwm_channel:= pinPWMTemp.byChannel, 
													frequency:= pinPWMTemp.wFrequency,
													polarity:= pinPWMTemp.bPolarity,
													diag_margin:= pinPWMTemp.bDiagMargin,
													safety_conf:= 0);		
								
	IF(pinPWMTemp.stInitError <> lib500_types.IO_ERRORTYPE.IO_E_OK) THEN initializePinError:= pinPWMTemp.stInitError; END_IF		
	pinPWMTemp.bInitialized:= (pinPWMTemp.stInitError = lib500_types.IO_ERRORTYPE.IO_E_OK);		
	IF NOT pinPWMTemp.bInitialized THEN initializeIO:= FALSE; END_IF
	
	paAllPWMOutputs[iPWMIterator]^:= pinPWMTemp;
	
END_FOR



FOR iPWDIterator:= 0 TO iAllPWDCursor - 1 BY 1 DO
	IF paAllPWDInputs[iPWDIterator] = 0 THEN CONTINUE; END_IF
	pinPWDTemp:= paAllPWDInputs[iPWDIterator]^;
	IF pinPWDTemp.bInitialized OR pinPWDTemp.byMinTTCModel > byTTCModel THEN CONTINUE; END_IF
	
	IF pinPWDTemp.readMode = pwdReadMode.incremental THEN
		pinPWDTemp.stInitError:= lib500.IO_PWD_IncInit(
												inc_channel:= pinPWDTemp.byChannel,
												mode:= pinPWDTemp.pwdMode,
												pupd:= pinPWDTemp.byPullType,
												count_init:= pinPWDTemp.wCountInit,
												safety_conf:= 0
								);	
								
	ELSIF pinPWDTemp.readMode = pwdReadMode.complex THEN	
		pinPWDTemp.stInitError:= lib500.IO_PWD_ComplexInit(
			timer_channel:= pinPWDTemp.byChannel, 
			pulse_mode:= pinPwdTemp.pulseMode, 
			freq_mode:= pinPWDTemp.freqMode, 
			capture_count:= pinPWDTemp.byCaptureCount, 
			pupd:= pinPWDTemp.byPullType, 
			safety_conf:= 0
		);
	
	END_IF
								
	IF(pinPWDTemp.stInitError <> lib500_types.IO_ERRORTYPE.IO_E_OK) THEN initializePinError:= pinPWDTemp.stInitError; END_IF	
	pinPWDTemp.bInitialized:= (pinPWDTemp.stInitError = lib500_types.IO_ERRORTYPE.IO_E_OK);		
	IF NOT pinPWDTemp.bInitialized THEN initializeIO:= FALSE; END_IF
	
	paAllPWDInputs[iPWDIterator]^:= pinPWDTemp;

END_FOR



FOR iPVGIterator:= 0 TO iAllPWDCursor - 1 BY 1 DO
	IF paAllPVGOutputs[iPVGIterator] = 0 THEN CONTINUE; END_IF
	pinPVGTemp:= paAllPVGOutputs[iPVGIterator]^;
	IF pinPVGTemp.bInitialized OR pinPVGTemp.byMinTTCModel > byTTCModel THEN CONTINUE; END_IF

	pinPVGTemp.stInitError:= lib500.IO_PVG_Init(pvg_channel:= pinPVGTemp.byChannel, output_value:= pinPVGTemp.wValue);
								
	IF(pinPVGTemp.stInitError <> lib500_types.IO_ERRORTYPE.IO_E_OK) THEN initializePinError:= pinPVGTemp.stInitError; END_IF	
	pinPVGTemp.bInitialized:= (pinPVGTemp.stInitError = lib500_types.IO_ERRORTYPE.IO_E_OK);		
	IF NOT pinPVGTemp.bInitialized THEN initializeIO:= FALSE; END_IF

	paAllPVGOutputs[iPVGIterator]^:= pinPVGTemp;

END_FOR



FOR iVOUTIterator:= 0 TO iAllVOUTCursor - 1 BY 1 DO
	IF paAllVOUTOutputs[iVOUTIterator] = 0 THEN CONTINUE; END_IF
	pinVOUTTemp:= paAllVOUTOutputs[iVOUTIterator]^;
	IF pinVOUTTemp.bInitialized OR pinVOUTTemp.byMinTTCModel > byTTCModel THEN CONTINUE; END_IF
	
	pinVOUTTemp.stInitError:= lib500.IO_VOUT_Init(vout_channel:= pinVOUTTemp.byChannel);	
								
	IF(pinVOUTTemp.stInitError <> lib500_types.IO_ERRORTYPE.IO_E_OK) THEN initializePinError:= pinVOUTTemp.stInitError; END_IF	
	pinVOUTTemp.bInitialized:= (pinVOUTTemp.stInitError = lib500_types.IO_ERRORTYPE.IO_E_OK);		
	IF NOT pinVOUTTemp.bInitialized THEN initializeIO:= FALSE; END_IF
	
	paAllVOUTOutputs[iVOUTIterator]^:= pinVOUTTemp;

END_FOR
END_METHOD

METHOD PUBLIC instantiateDO
VAR_INPUT
	outPointer: POINTER TO pinDIO;
	byChannel: BYTE;
END_VAR
instantiateDIO(outPointer, byChannel, 0);

paAllDigitalOutputs[iAllDOCursor]:= outPointer;
iAllDOCursor:= iAllDOCursor + 1;

IF iAllDOCursor >= DO_maxIndex THEN
	iAllDOCursor:= 0;
END_IF
END_METHOD

METHOD PRIVATE instantiateDIO
VAR_INPUT
	outPointer: POINTER TO pinDIO;
	byChannel: BYTE;
	byPullType: BYTE:= 0;
END_VAR
outPointer^.byChannel:= byChannel;
outPointer^.byPullType:= byPullType;
END_METHOD

METHOD PUBLIC instantiatePVG
VAR_INPUT
	outPointer: POINTER TO pinPVG;
	byChannel: BYTE;
	wValue: WORD:= 5000;
END_VAR
outPointer^.byChannel:= byChannel;
outPointer^.wValue:= wValue;

paAllPVGOutputs[iAllPWDCursor]:= outPointer;
iAllPVGCursor:= iAllPVGCursor + 1;

IF iAllPVGCursor >= PVG_maxIndex THEN
	iAllPVGCursor:= 0;
END_IF
END_METHOD

METHOD setOutputs : BOOL
VAR
	iPowerIterator: INT;
	iDIOterator: INT;
	iPWMIterator: INT;
	iVOUTIterator: INT;
	iPVGIterator: INT;
	
	pinPowerTemp: pinPower;
	pinDOTemp: pinDIO;
	pinPWMTemp: pinPWM;
	pinVOUTTemp: pinVOUT;
	pinPVGTemp: pinPVG;
END_VAR
setOutputs:= TRUE;
outputPinError:= lib500_types.IO_ERRORTYPE.IO_E_OK;

FOR iPowerIterator:= 0 TO iAllPowerCursor - 1 BY 1 DO
	IF paAllPowerOutputs[iPowerIterator] = 0 THEN CONTINUE; END_IF
	pinPowerTemp:= paAllPowerOutputs[iPowerIterator]^;
	IF NOT pinPowerTemp.bInitialized OR pinPowerTemp.byMinTTCModel > byTTCModel THEN CONTINUE; END_IF
	
	pinPowerTemp.stError:= lib500.IO_POWER_Set(
								pin:= pinPowerTemp.byChannel,
								mode:= pinPowerTemp.mode
							);		
		
								
	IF (pinPowerTemp.stError <> lib500_types.IO_ERRORTYPE.IO_E_OK AND pinPowerTemp.stError <> lib500_types.IO_ERRORTYPE.IO_E_NO_DIAG) THEN 
		setOutputs:= FALSE; 
		outputPinError:= pinPowerTemp.stError;
	END_IF		
	
	paAllPowerOutputs[iPowerIterator]^:= pinPowerTemp;	
END_FOR

FOR iDIOterator:= 0 TO iAllDOCursor - 1 BY 1 DO	
	IF paAllDigitalOutputs[iDIOterator] = 0 THEN CONTINUE; END_IF
	pinDOTemp:= paAllDigitalOutputs[iDIOterator]^;
	IF NOT pinDOTemp.bInitialized OR pinDOTemp.byMinTTCModel > byTTCModel THEN CONTINUE; END_IF
	
	pinDOTemp.stError:= lib500.IO_DO_Set(do_channel:= pinDOTemp.byChannel, do_value:= pinDOTemp.bValue);		
													
	pinDOTemp.stErrorGetCut:= lib500.IO_DO_GetCur(do_channel:= pinDOTemp.byChannel, 
													current:= ADR(pinDOTemp.wCurrent),
													fresh:= ADR(pinDOTemp.bCurrentFresh));		
																	
	IF pinDOTemp.stError = lib500_types.IO_ERRORTYPE.IO_E_FET_PROT_REENABLE THEN
		lib500.IO_DO_ResetProtection(do_channel:= pinDOTemp.byChannel, ADR(pinPowerTemp.byResetCount));
	END_IF
	IF pinDOTemp.stError <> lib500_types.IO_ERRORTYPE.IO_E_OK AND pinDOTemp.stError <> lib500_types.IO_ERRORTYPE.IO_E_NO_DIAG AND pinDOTemp.stError <> lib500_types.IO_ERRORTYPE.IO_E_OPEN_LOAD THEN 
		setOutputs:= FALSE; 
		outputPinError:= pinDOTemp.stError;
	END_IF		
	IF pinDOTemp.stErrorGetCut <> lib500_types.IO_ERRORTYPE.IO_E_OK  AND pinDOTemp.stError <> lib500_types.IO_ERRORTYPE.IO_E_NO_DIAG THEN 
		setOutputs:= FALSE; 
		outputPinError:= pinDOTemp.stErrorGetCut;
	END_IF		
							
	paAllDigitalOutputs[iDIOterator]^:= pinDOTemp;	
END_FOR


FOR iPWMIterator:= 0 TO iAllPWMCursor - 1 BY 1 DO
	IF paAllPWMOutputs[iPWMIterator] = 0 THEN CONTINUE; END_IF
	pinPWMTemp:= paAllPWMOutputs[iPWMIterator]^;
	IF NOT pinPWMTemp.bInitialized OR pinPWMTemp.byMinTTCModel > byTTCModel THEN CONTINUE; END_IF
	
	pinPWMTemp.stError:= lib500.IO_PWM_SetDuty(pwm_channel:= pinPWMTemp.byChannel, 
													duty_cycle:= pinPWMTemp.wDuty,
													high_time_fb:= ADR(pinPWMTemp.wFeedbackHighTime),
													period_fb:= ADR(pinPWMTemp.wPeriodFeedback));
													
	pinPWMTemp.stErrorGetCut:= lib500.IO_PWM_GetCur(pwm_channel:= pinPWMTemp.byChannel, 
													current:= ADR(pinPWMTemp.wCurrent),
													fresh:= ADR(pinPWMTemp.bCurrentFresh));		
		
	IF pinPWMTemp.stError = lib500_types.IO_ERRORTYPE.IO_E_FET_PROT_REENABLE THEN
		lib500.IO_PWM_ResetProtection(pwm_channel:= pinPWMTemp.byChannel, ADR(pinPowerTemp.byResetCount));
	END_IF
	
	IF (pinPWMTemp.stError <> lib500_types.IO_ERRORTYPE.IO_E_OK AND pinPWMTemp.stError <> lib500_types.IO_ERRORTYPE.IO_E_NO_DIAG) THEN
		setOutputs:= FALSE; 
		outputPinError:= pinPWMTemp.stError;
	END_IF
	IF pinPWMTemp.stErrorGetCut <> lib500_types.IO_ERRORTYPE.IO_E_OK AND pinPWMTemp.stError <> lib500_types.IO_ERRORTYPE.IO_E_NO_DIAG THEN 
		setOutputs:= FALSE; 
		outputPinError:= pinPWMTemp.stErrorGetCut;
	END_IF		
	
	paAllPWMOutputs[iPWMIterator]^:= pinPWMTemp;	
END_FOR


FOR iVOUTIterator:= 0 TO iAllVOUTCursor - 1 BY 1 DO
	IF paAllVOUTOutputs[iVOUTIterator] = 0 THEN CONTINUE; END_IF
	pinVOUTTemp:= paAllVOUTOutputs[iVOUTIterator]^;
	IF NOT pinVOUTTemp.bInitialized OR pinVOUTTemp.byMinTTCModel > byTTCModel THEN CONTINUE; END_IF
	
	pinVOUTTemp.stError:= lib500.IO_VOUT_SetVoltage(
								vout_channel:= pinVOUTTemp.byChannel,
								output_voltage:= pinVOUTTemp.wOutputVoltageMv
							);		
		
	IF (pinVOUTTemp.stError <> lib500_types.IO_ERRORTYPE.IO_E_OK AND pinVOUTTemp.stError <> lib500_types.IO_ERRORTYPE.IO_E_NO_DIAG) THEN 
		setOutputs:= FALSE; 
		outputPinError:= pinVOUTTemp.stError;
	END_IF		
	
	paAllVOUTOutputs[iVOUTIterator]^:= pinVOUTTemp;	
END_FOR


FOR iPVGIterator:= 0 TO iAllPVGCursor - 1 BY 1 DO
	IF paAllPVGOutputs[iPVGIterator] = 0 THEN CONTINUE; END_IF
	pinPVGTemp:= paAllPVGOutputs[iPVGIterator]^;
	IF NOT pinPVGTemp.bInitialized OR pinPVGTemp.byMinTTCModel > byTTCModel THEN CONTINUE; END_IF
	
